gfCNCPoint1[4843] = {X 83.0240, Y 40.8731, Z -1.3333, A 0.000, B 0.000, C 0.000 }
gfCNCPoint1[4844] = {X 83.0237, Y 16.3120, Z -1.3333, A 0.000, B 0.000, C 0.000 }
gfCNCPoint1[4845] = {X 82.3786, Y 15.6228, Z -1.3333, A 0.000, B 0.000, C 0.000 }
gfCNCPoint1[4846] = {X 81.8954, Y 14.8118, Z -1.3333, A 0.000, B 0.000, C 0.000 }
gfCNCPoint1[4847] = {X 81.5963, Y 13.9165, Z -1.3333, A 0.000, B 0.000, C 0.000 }
gfCNCPoint1[4848] = {X 81.4951, Y 12.9779, Z -1.3333, A 0.000, B 0.000, C 0.000 }
gfCNCPoint1[4849] = {X 81.4951, Y 12.1868, Z -1.3333, A 0.000, B 0.000, C 0.000 }
gfCNCPoint1[4850] = {X 81.5776, Y 11.3388, Z -1.3333, A 0.000, B 0.000, C 0.000 }
gfCNCPoint1[4851] = {X 81.8219, Y 10.5227, Z -1.3333, A 0.000, B 0.000, C 0.000 }
gfCNCPoint1[4852] = {X 82.2190, Y 9.7689, Z -1.3333, A 0.000, B 0.000, C 0.000 }
gfCNCPoint1[4853] = {X 81.8180, Y 9.5051, Z -1.3333, A 0.000, B 0.000, C 0.000 }
gfCNCPoint1[4854] = {X 68.9232, Y 9.5051, Z -1.3333, A 0.000, B 0.000, C 0.000 }
gfCNCPoint1[4855] = {X 69.1905, Y 10.7210, Z -1.3333, A 0.000, B 0.000, C 0.000 }
gfCNCPoint1[4856] = {X 69.2995, Y 11.9611, Z -1.3333, A 0.000, B 0.000, C 0.000 }
gfCNCPoint1[4857] = {X 69.3015, Y 12.0739, Z -1.3333, A 0.000, B 0.000, C 0.000 }
gfCNCPoint1[4858] = {X 69.3021, Y 12.1868, Z -1.3333, A 0.000, B 0.000, C 0.000 }
gfCNCPoint1[4859] = {X 69.3017, Y 13.0686, Z -1.3333, A 0.000, B 0.000, C 0.000 }
gfCNCPoint1[4860] = {X 69.2131, Y 14.2875, Z -1.3333, A 0.000, B 0.000, C 0.000 }
gfCNCPoint1[4861] = {X 68.9717, Y 15.4855, Z -1.3333, A 0.000, B 0.000, C 0.000 }
gfCNCPoint1[4862] = {X 73.2474, Y 26.9301, Z -1.3333, A 0.000, B 0.000, C 0.000 }
gfCNCPoint1[4863] = {X 77.7438, Y 25.2502, Z -1.3333, A 0.000, B 0.000, C 0.000 }
gfCNCPoint1[4864] = {X 77.7437, Y 18.1989, Z -1.3333, A 0.000, B 0.000, C 0.000 }
gfCNCPoint1[4865] = {X 77.0787, Y 16.9748, Z -1.3333, A 0.000, B 0.000, C 0.000 }
gfCNCPoint1[4866] = {X 76.5963, Y 15.6678, Z -1.3333, A 0.000, B 0.000, C 0.000 }
gfCNCPoint1[4867] = {X 76.3065, Y 14.3051, Z -1.3333, A 0.000, B 0.000, C 0.000 }
gfCNCPoint1[4868] = {X 74.0412, Y 14.3051, Z -1.3333, A 0.000, B 0.000, C 0.000 }
gfCNCPoint1[4869] = {X 73.9997, Y 14.6975, Z -1.3333, A 0.000, B 0.000, C 0.000 }
gfCNCPoint1[4870] = {X 73.9475, Y 15.0886, Z -1.3333, A 0.000, B 0.000, C 0.000 }
gfCNCPoint1[4871] = {X 77.7438, Y 25.2502, Z -1.3333, A 0.000, B 0.000, C 0.000 }
gfCNCPoint1[4872] = {X 75.4956, Y 26.0902, Z -1.3333, A 0.000, B 0.000, C 0.000 }
gfCNCPoint1[4873] = {X 78.9539, Y 35.3470, Z -1.3333, A 0.000, B 0.000, C 0.000 }
gfCNCPoint1[4874] = {X 79.5719, Y 35.9625, Z -1.3333, A 0.000, B 0.000, C 0.000 }
gfCNCPoint1[4875] = {X 80.1440, Y 36.6209, Z -1.3333, A 0.000, B 0.000, C 0.000 }
gfCNCPoint1[4876] = {X 80.1437, Y 17.4412, Z -1.3333, A 0.000, B 0.000, C 0.000 }
gfCNCPoint1[4877] = {X 79.4950, Y 16.4475, Z -1.3333, A 0.000, B 0.000, C 0.000 }
gfCNCPoint1[4878] = {X 79.0163, Y 15.3615, Z -1.3333, A 0.000, B 0.000, C 0.000 }
gfCNCPoint1[4879] = {X 78.7204, Y 14.2122, Z -1.3333, A 0.000, B 0.000, C 0.000 }
gfCNCPoint1[4880] = {X 78.6153, Y 13.0301, Z -1.3333, A 0.000, B 0.000, C 0.000 }
gfCNCPoint1[4881] = {X 78.6151, Y 12.1868, Z -1.3333, A 0.000, B 0.000, C 0.000 }
gfCNCPoint1[4882] = {X 78.6164, Y 12.0459, Z -1.3333, A 0.000, B 0.000, C 0.000 }
gfCNCPoint1[4883] = {X 78.6205, Y 11.9051, Z -1.3333, A 0.000, B 0.000, C 0.000 }
gfCNCPoint1[4884] = {X 71.6988, Y 11.9051, Z -1.3333, A 0.000, B 0.000, C 0.000 }
gfCNCPoint1[4885] = {X 71.7013, Y 12.0460, Z -1.3333, A 0.000, B 0.000, C 0.000 }
gfCNCPoint1[4886] = {X 71.7021, Y 12.1868, Z -1.3333, A 0.000, B 0.000, C 0.000 }
gfCNCPoint1[4887] = {X 71.7016, Y 13.0911, Z -1.3333, A 0.000, B 0.000, C 0.000 }
gfCNCPoint1[4888] = {X 71.6389, Y 14.2118, Z -1.3333, A 0.000, B 0.000, C 0.000 }
gfCNCPoint1[4889] = {X 71.4726, Y 15.3218, Z -1.3333, A 0.000, B 0.000, C 0.000 }
gfCNCPoint1[4890] = {X 75.4956, Y 26.0902, Z -1.3333, A 0.000, B 0.000, C 0.000 }
gfCNCPoint1[4891] = {X 73.2474, Y 26.9301, Z -1.3333, A 0.000, B 0.000, C 0.000 }
gfCNCPoint1[4892] = {X 76.9168, Y 36.7519, Z -1.3333, A 0.000, B 0.000, C 0.000 }
gfCNCPoint1[4893] = {X 77.6311, Y 37.4061, Z -1.3333, A 0.000, B 0.000, C 0.000 }
gfCNCPoint1[4894] = {X 78.2765, Y 38.1284, Z -1.3333, A 0.000, B 0.000, C 0.000 }
gfCNCPoint1[4895] = {X 79.0237, Y 39.1932, Z -1.3333, A 0.000, B 0.000, C 0.000 }
gfCNCPoint1[4896] = {X 79.6214, Y 40.3484, Z -1.3333, A 0.000, B 0.000, C 0.000 }
gfCNCPoint1[4897] = {X 80.0588, Y 41.5734, Z -1.3333, A 0.000, B 0.000, C 0.000 }
gfCNCPoint1[4898] = {X 80.3281, Y 42.8460, Z -1.3333, A 0.000, B 0.000, C 0.000 }
gfCNCPoint1[4899] = {X 80.4242, Y 44.1432, Z -1.3333, A 0.000, B 0.000, C 0.000 }
gfCNCPoint1[4900] = {X 80.4245, Y 45.0000, Z -1.3333, A 0.000, B 0.000, C 0.000 }
gfCNCPoint1[4901] = {X 80.3511, Y 46.1898, Z -1.3333, A 0.000, B 0.000, C 0.000 }
gfCNCPoint1[4902] = {X 80.1320, Y 47.3615, Z -1.3333, A 0.000, B 0.000, C 0.000 }
gfCNCPoint1[4903] = {X 79.7706, Y 48.4974, Z -1.3333, A 0.000, B 0.000, C 0.000 }
gfCNCPoint1[4904] = {X 79.2722, Y 49.5803, Z -1.3333, A 0.000, B 0.000, C 0.000 }
gfCNCPoint1[4905] = {X 78.4688, Y 50.8341, Z -1.3333, A 0.000, B 0.000, C 0.000 }
gfCNCPoint1[4906] = {X 77.4826, Y 51.9498, Z -1.3333, A 0.000, B 0.000, C 0.000 }
gfCNCPoint1[4907] = {X 76.3369, Y 52.9011, Z -1.3333, A 0.000, B 0.000, C 0.000 }
gfCNCPoint1[4908] = {X 75.0589, Y 53.6653, Z -1.3333, A 0.000, B 0.000, C 0.000 }
gfCNCPoint1[4909] = {X 73.6787, Y 54.2246, Z -1.3333, A 0.000, B 0.000, C 0.000 }
gfCNCPoint1[4910] = {X 72.2292, Y 54.5655, Z -1.3333, A 0.000, B 0.000, C 0.000 }
gfCNCPoint1[4911] = {X 70.7445, Y 54.6800, Z -1.3333, A 0.000, B 0.000, C 0.000 }
gfCNCPoint1[4912] = {X 64.1851, Y 54.6800, Z -1.3333, A 0.000, B 0.000, C 0.000 }
gfCNCPoint1[4913] = {X 62.7229, Y 54.5689, Z -1.3333, A 0.000, B 0.000, C 0.000 }
gfCNCPoint1[4914] = {X 61.2943, Y 54.2383, Z -1.3333, A 0.000, B 0.000, C 0.000 }
gfCNCPoint1[4915] = {X 59.9320, Y 53.6956, Z -1.3333, A 0.000, B 0.000, C 0.000 }
gfCNCPoint1[4916] = {X 58.6673, Y 52.9534, Z -1.3333, A 0.000, B 0.000, C 0.000 }
gfCNCPoint1[4917] = {X 57.5293, Y 52.0286, Z -1.3333, A 0.000, B 0.000, C 0.000 }
gfCNCPoint1[4918] = {X 56.6337, Y 51.0563, Z -1.3333, A 0.000, B 0.000, C 0.000 }
gfCNCPoint1[4919] = {X 55.8790, Y 49.9710, Z -1.3333, A 0.000, B 0.000, C 0.000 }
gfCNCPoint1[4920] = {X 55.1243, Y 51.0563, Z -1.3333, A 0.000, B 0.000, C 0.000 }
gfCNCPoint1[4921] = {X 54.2288, Y 52.0286, Z -1.3333, A 0.000, B 0.000, C 0.000 }
gfCNCPoint1[4922] = {X 53.0907, Y 52.9534, Z -1.3333, A 0.000, B 0.000, C 0.000 }
gfCNCPoint1[4923] = {X 51.8261, Y 53.6956, Z -1.3333, A 0.000, B 0.000, C 0.000 }
gfCNCPoint1[4924] = {X 50.4638, Y 54.2383, Z -1.3333, A 0.000, B 0.000, C 0.000 }
gfCNCPoint1[4925] = {X 49.0351, Y 54.5689, Z -1.3333, A 0.000, B 0.000, C 0.000 }
gfCNCPoint1[4926] = {X 47.5729, Y 54.6800, Z -1.3333, A 0.000, B 0.000, C 0.000 }
gfCNCPoint1[4927] = {X 40.6393, Y 54.6800, Z -1.3333, A 0.000, B 0.000, C 0.000 }
gfCNCPoint1[4928] = {X 39.2448, Y 54.5790, Z -1.3333, A 0.000, B 0.000, C 0.000 }
gfCNCPoint1[4929] = {X 37.8793, Y 54.2782, Z -1.3333, A 0.000, B 0.000, C 0.000 }
gfCNCPoint1[4930] = {X 36.5715, Y 53.7838, Z -1.3333, A 0.000, B 0.000, C 0.000 }
gfCNCPoint1[4931] = {X 35.3485, Y 53.1062, Z -1.3333, A 0.000, B 0.000, C 0.000 }
gfCNCPoint1[4932] = {X 33.9156, Y 54.1337, Z -1.3333, A 0.000, B 0.000, C 0.000 }
gfCNCPoint1[4933] = {X 32.3650, Y 54.9732, Z -1.3333, A 0.000, B 0.000, C 0.000 }
gfCNCPoint1[4934] = {X 30.7213, Y 55.6115, Z -1.3333, A 0.000, B 0.000, C 0.000 }
gfCNCPoint1[4935] = {X 29.0105, Y 56.0384, Z -1.3333, A 0.000, B 0.000, C 0.000 }
gfCNCPoint1[4936] = {X 27.2597, Y 56.2471, Z -1.3333, A 0.000, B 0.000, C 0.000 }
gfCNCPoint1[4937] = {X 25.4108, Y 57.0591, Z -1.3333, A 0.000, B 0.000, C 0.000 }
gfCNCPoint1[4938] = {X 23.5216, Y 57.7721, Z -1.3333, A 0.000, B 0.000, C 0.000 }
gfCNCPoint1[4939] = {X 21.5973, Y 58.3841, Z -1.3333, A 0.000, B 0.000, C 0.000 }
gfCNCPoint1[4940] = {X 21.0307, Y 58.5413, Z -1.3333, A 0.000, B 0.000, C 0.000 }
gfCNCPoint1[4941] = {X 18.7673, Y 59.0805, Z -1.3333, A 0.000, B 0.000, C 0.000 }
gfCNCPoint1[4942] = {X 16.4706, Y 59.4536, Z -1.3333, A 0.000, B 0.000, C 0.000 }
gfCNCPoint1[4943] = {X 14.1529, Y 59.6585, Z -1.3333, A 0.000, B 0.000, C 0.000 }
gfCNCPoint1[4944] = {X 11.8264, Y 59.6941, Z -1.3333, A 0.000, B 0.000, C 0.000 }
gfCNCPoint1[4945] = {X 9.5035, Y 59.5603, Z -1.3333, A 0.000, B 0.000, C 0.000 }
gfCNCPoint1[4946] = {X 9.5035, Y 90.4949, Z -1.3333, A 0.000, B 0.000, C 0.000 }
gfCNCPoint1[4947] = {X 114.8635, Y 90.4949, Z -1.3333, A 0.000, B 0.000, C 0.000 }
gfCNCPoint1[4948] = {X 115.7480, Y 89.2990, Z -1.3333, A 0.000, B 0.000, C 0.000 }
gfCNCPoint1[4949] = {X 116.7726, Y 88.2208, Z -1.3333, A 0.000, B 0.000, C 0.000 }
gfCNCPoint1[4950] = {X 117.9221, Y 87.2767, Z -1.3333, A 0.000, B 0.000, C 0.000 }
gfCNCPoint1[4951] = {X 119.1788, Y 86.4811, Z -1.3333, A 0.000, B 0.000, C 0.000 }
gfCNCPoint1[4952] = {X 120.5238, Y 85.8459, Z -1.3333, A 0.000, B 0.000, C 0.000 }
gfCNCPoint1[4953] = {X 121.9366, Y 85.3808, Z -1.3333, A 0.000, B 0.000, C 0.000 }
gfCNCPoint1[4954] = {X 123.3959, Y 85.0929, Z -1.3333, A 0.000, B 0.000, C 0.000 }
gfCNCPoint1[4955] = {X 123.5628, Y 84.9132, Z -1.3333, A 0.000, B 0.000, C 0.000 }
gfCNCPoint1[4956] = {X 123.7278, Y 84.7318, Z -1.3333, A 0.000, B 0.000, C 0.000 }
gfCNCPoint1[4957] = {X 147.2181, Y 58.9362, Z -1.3333, A 0.000, B 0.000, C 0.000 }
gfCNCPoint1[4958] = {X 147.2180, Y 58.0000, Z -1.3333, A 0.000, B 0.000, C 0.000 }
gfCNCPoint1[4959] = {X 147.2987, Y 56.6058, Z -1.3333, A 0.000, B 0.000, C 0.000 }
gfCNCPoint1[4960] = {X 147.5398, Y 55.2303, Z -1.3333, A 0.000, B 0.000, C 0.000 }
gfCNCPoint1[4961] = {X 148.0022, Y 53.7185, Z -1.3333, A 0.000, B 0.000, C 0.000 }
gfCNCPoint1[4962] = {X 148.6580, Y 52.2800, Z -1.3333, A 0.000, B 0.000, C 0.000 }
gfCNCPoint1[4963] = {X 143.0396, Y 52.2800, Z -1.3333, A 0.000, B 0.000, C 0.000 }
gfCNCPoint1[4964] = {X 141.7807, Y 52.1703, Z -1.3333, A 0.000, B 0.000, C 0.000 }
gfCNCPoint1[4965] = {X 140.5597, Y 51.8446, Z -1.3333, A 0.000, B 0.000, C 0.000 }
gfCNCPoint1[4966] = {X 139.4134, Y 51.3126, Z -1.3333, A 0.000, B 0.000, C 0.000 }
gfCNCPoint1[4967] = {X 138.3764, Y 50.5904, Z -1.3333, A 0.000, B 0.000, C 0.000 }
gfCNCPoint1[4968] = {X 137.4799, Y 49.6998, Z -1.3333, A 0.000, B 0.000, C 0.000 }
gfCNCPoint1[4969] = {X 136.7509, Y 48.6675, Z -1.3333, A 0.000, B 0.000, C 0.000 }
gfCNCPoint1[4970] = {X 136.2114, Y 47.5248, Z -1.3333, A 0.000, B 0.000, C 0.000 }
gfCNCPoint1[4971] = {X 135.8777, Y 46.3059, Z -1.3333, A 0.000, B 0.000, C 0.000 }
gfCNCPoint1[4972] = {X 135.7598, Y 45.0477, Z -1.3333, A 0.000, B 0.000, C 0.000 }
gfCNCPoint1[4973] = {X 135.7601, Y 44.1247, Z -1.3333, A 0.000, B 0.000, C 0.000 }
gfCNCPoint1[4974] = {X 135.8408, Y 43.1249, Z -1.3333, A 0.000, B 0.000, C 0.000 }
gfCNCPoint1[4975] = {X 136.0581, Y 42.1457, Z -1.3333, A 0.000, B 0.000, C 0.000 }
gfCNCPoint1[4976] = {X 138.3597, Y 42.8258, Z -1.3333, A 0.000, B 0.000, C 0.000 }
gfCNCPoint1[4977] = {X 138.6721, Y 42.0319, Z -1.3333, A 0.000, B 0.000, C 0.000 }
gfCNCPoint1[4978] = {X 139.1179, Y 41.3046, Z -1.3333, A 0.000, B 0.000, C 0.000 }
gfCNCPoint1[4979] = {X 139.6836, Y 40.6660, Z -1.3333, A 0.000, B 0.000, C 0.000 }
gfCNCPoint1[4980] = {X 139.6836, Y 20.4363, Z -1.3333, A 0.000, B 0.000, C 0.000 }
gfCNCPoint1[4981] = {X 137.7113, Y 20.4357, Z -1.3333, A 0.000, B 0.000, C 0.000 }
gfCNCPoint1[4982] = {X 137.0006, Y 21.1817, Z -1.3333, A 0.000, B 0.000, C 0.000 }
gfCNCPoint1[4983] = {X 136.1491, Y 21.7619, Z -1.3333, A 0.000, B 0.000, C 0.000 }
gfCNCPoint1[4984] = {X 135.4282, Y 22.0767, Z -1.3333, A 0.000, B 0.000, C 0.000 }
gfCNCPoint1[4985] = {X 134.6660, Y 22.2715, Z -1.3333, A 0.000, B 0.000, C 0.000 }
gfCNCPoint1[4986] = {X 133.8824, Y 22.3414, Z -1.3333, A 0.000, B 0.000, C 0.000 }
gfCNCPoint1[4987] = {X 133.2006, Y 22.3415, Z -1.3333, A 0.000, B 0.000, C 0.000 }
gfCNCPoint1[4988] = {X 132.2486, Y 22.2478, Z -1.3333, A 0.000, B 0.000, C 0.000 }
gfCNCPoint1[4989] = {X 131.3331, Y 21.9701, Z -1.3333, A 0.000, B 0.000, C 0.000 }
gfCNCPoint1[4990] = {X 130.4895, Y 21.5191, Z -1.3333, A 0.000, B 0.000, C 0.000 }
gfCNCPoint1[4991] = {X 129.7500, Y 20.9122, Z -1.3333, A 0.000, B 0.000, C 0.000 }
gfCNCPoint1[4992] = {X 129.1431, Y 20.1727, Z -1.3333, A 0.000, B 0.000, C 0.000 }
gfCNCPoint1[4993] = {X 128.6921, Y 19.3290, Z -1.3333, A 0.000, B 0.000, C 0.000 }
gfCNCPoint1[4994] = {X 128.4144, Y 18.4136, Z -1.3333, A 0.000, B 0.000, C 0.000 }
gfCNCPoint1[4995] = {X 128.3206, Y 17.4615, Z -1.3333, A 0.000, B 0.000, C 0.000 }
gfCNCPoint1[4996] = {X 128.3206, Y 10.4835, Z -1.3333, A 0.000, B 0.000, C 0.000 }
gfCNCPoint1[4997] = {X 128.3317, Y 10.1548, Z -1.3333, A 0.000, B 0.000, C 0.000 }
gfCNCPoint1[4998] = {X 128.3649, Y 9.8277, Z -1.3333, A 0.000, B 0.000, C 0.000 }
gfCNCPoint1[4999] = {X 128.6078, Y 8.8342, Z -1.3333, A 0.000, B 0.000, C 0.000 }
gfCNCPoint1[5000] = {X 129.0524, Y 7.9132, Z -1.3333, A 0.000, B 0.000, C 0.000 }
gfCNCPoint1[5001] = {X 129.6792, Y 7.1051, Z -1.3333, A 0.000, B 0.000, C 0.000 }
gfCNCPoint1[5002] = {X 130.0255, Y 7.4374, Z -1.3333, A 0.000, B 0.000, C 0.000 }
gfCNCPoint1[5003] = {X 130.6996, Y 6.8635, Z -1.3333, A 0.000, B 0.000, C 0.000 }
gfCNCPoint1[5004] = {X 131.4748, Y 6.4361, Z -1.3333, A 0.000, B 0.000, C 0.000 }
gfCNCPoint1[5005] = {X 132.3199, Y 6.1726, Z -1.3333, A 0.000, B 0.000, C 0.000 }
gfCNCPoint1[5006] = {X 133.2007, Y 6.0835, Z -1.3333, A 0.000, B 0.000, C 0.000 }
gfCNCPoint1[5007] = {X 133.8874, Y 6.0837, Z -1.3333, A 0.000, B 0.000, C 0.000 }
gfCNCPoint1[5008] = {X 134.7192, Y 6.1718, Z -1.3333, A 0.000, B 0.000, C 0.000 }
gfCNCPoint1[5009] = {X 135.5192, Y 6.4156, Z -1.3333, A 0.000, B 0.000, C 0.000 }
gfCNCPoint1[5010] = {X 136.2587, Y 6.8064, Z -1.3333, A 0.000, B 0.000, C 0.000 }
gfCNCPoint1[5011] = {X 136.9108, Y 7.3301, Z -1.3333, A 0.000, B 0.000, C 0.000 }
gfCNCPoint1[5012] = {X 137.4521, Y 7.9677, Z -1.3333, A 0.000, B 0.000, C 0.000 }
gfCNCPoint1[5013] = {X 155.0706, Y 7.9677, Z -1.3333, A 0.000, B 0.000, C 0.000 }
gfCNCPoint1[5014] = {X 155.6184, Y 7.3238, Z -1.3333, A 0.000, B 0.000, C 0.000 }
gfCNCPoint1[5015] = {X 156.2792, Y 6.7965, Z -1.3333, A 0.000, B 0.000, C 0.000 }
gfCNCPoint1[5016] = {X 157.0287, Y 6.4053, Z -1.3333, A 0.000, B 0.000, C 0.000 }
gfCNCPoint1[5017] = {X 157.8391, Y 6.1647, Z -1.3333, A 0.000, B 0.000, C 0.000 }
gfCNCPoint1[5018] = {X 158.6806, Y 6.0835, Z -1.3333, A 0.000, B 0.000, C 0.000 }
gfCNCPoint1[5019] = {X 159.3791, Y 6.0839, Z -1.3333, A 0.000, B 0.000, C 0.000 }
gfCNCPoint1[5020] = {X 160.3488, Y 6.2050, Z -1.3333, A 0.000, B 0.000, C 0.000 }
gfCNCPoint1[5021] = {X 161.2678, Y 6.5371, Z -1.3333, A 0.000, B 0.000, C 0.000 }
gfCNCPoint1[5022] = {X 162.0908, Y 7.0639, Z -1.3333, A 0.000, B 0.000, C 0.000 }
gfCNCPoint1[5023] = {X 162.7773, Y 7.7593, Z -1.3333, A 0.000, B 0.000, C 0.000 }
gfCNCPoint1[5024] = {X 163.2934, Y 8.5891, Z -1.3333, A 0.000, B 0.000, C 0.000 }
gfCNCPoint1[5025] = {X 163.6136, Y 9.5124, Z -1.3333, A 0.000, B 0.000, C 0.000 }
gfCNCPoint1[5026] = {X 163.7221, Y 10.4835, Z -1.3333, A 0.000, B 0.000, C 0.000 }
gfCNCPoint1[5027] = {X 163.7221, Y 17.4615, Z -1.3333, A 0.000, B 0.000, C 0.000 }
gfCNCPoint1[5028] = {X 163.6118, Y 18.4406, Z -1.3333, A 0.000, B 0.000, C 0.000 }
gfCNCPoint1[5029] = {X 163.2863, Y 19.3706, Z -1.3333, A 0.000, B 0.000, C 0.000 }
gfCNCPoint1[5030] = {X 162.7621, Y 20.2049, Z -1.3333, A 0.000, B 0.000, C 0.000 }
gfCNCPoint1[5031] = {X 162.0654, Y 20.9016, Z -1.3333, A 0.000, B 0.000, C 0.000 }
gfCNCPoint1[5032] = {X 161.2312, Y 21.4258, Z -1.3333, A 0.000, B 0.000, C 0.000 }
gfCNCPoint1[5033] = {X 160.3011, Y 21.7512, Z -1.3333, A 0.000, B 0.000, C 0.000 }
gfCNCPoint1[5034] = {X 159.3221, Y 21.8615, Z -1.3333, A 0.000, B 0.000, C 0.000 }
gfCNCPoint1[5035] = {X 158.6785, Y 21.8615, Z -1.3333, A 0.000, B 0.000, C 0.000 }
gfCNCPoint1[5036] = {X 157.8332, Y 21.7759, Z -1.3333, A 0.000, B 0.000, C 0.000 }
gfCNCPoint1[5037] = {X 157.0197, Y 21.5308, Z -1.3333, A 0.000, B 0.000, C 0.000 }
gfCNCPoint1[5038] = {X 156.2678, Y 21.1352, Z -1.3333, A 0.000, B 0.000, C 0.000 }
gfCNCPoint1[5039] = {X 155.6049, Y 20.6037, Z -1.3333, A 0.000, B 0.000, C 0.000 }
gfCNCPoint1[5040] = {X 155.0555, Y 19.9556, Z -1.3333, A 0.000, B 0.000, C 0.000 }
gfCNCPoint1[5041] = {X 152.3555, Y 19.9571, Z -1.3333, A 0.000, B 0.000, C 0.000 }
gfCNCPoint1[5042] = {X 152.3538, Y 40.8427, Z -1.3333, A 0.000, B 0.000, C 0.000 }
gfCNCPoint1[5043] = {X 152.8077, Y 41.3321, Z -1.3333, A 0.000, B 0.000, C 0.000 }
gfCNCPoint1[5044] = {X 152.8988, Y 41.4411, Z -1.3333, A 0.000, B 0.000, C 0.000 }
gfCNCPoint1[5045] = {X 153.4331, Y 42.2816, Z -1.3333, A 0.000, B 0.000, C 0.000 }
gfCNCPoint1[5046] = {X 153.7667, Y 43.2199, Z -1.3333, A 0.000, B 0.000, C 0.000 }
gfCNCPoint1[5047] = {X 153.8831, Y 44.2089, Z -1.3333, A 0.000, B 0.000, C 0.000 }
gfCNCPoint1[5048] = {X 153.8829, Y 45.0423, Z -1.3333, A 0.000, B 0.000, C 0.000 }
gfCNCPoint1[5049] = {X 153.7646, Y 46.0144, Z -1.3333, A 0.000, B 0.000, C 0.000 }
gfCNCPoint1[5050] = {X 153.4342, Y 46.9363, Z -1.3333, A 0.000, B 0.000, C 0.000 }
gfCNCPoint1[5051] = {X 152.9080, Y 47.7622, Z -1.3333, A 0.000, B 0.000, C 0.000 }
gfCNCPoint1[5052] = {X 152.2123, Y 48.4513, Z -1.3333, A 0.000, B 0.000, C 0.000 }
gfCNCPoint1[5053] = {X 151.3813, Y 48.9695, Z -1.3333, A 0.000, B 0.000, C 0.000 }
gfCNCPoint1[5054] = {X 150.4563, Y 49.2910, Z -1.3333, A 0.000, B 0.000, C 0.000 }
gfCNCPoint1[5055] = {X 149.4831, Y 49.4000, Z -1.3333, A 0.000, B 0.000, C 0.000 }
gfCNCPoint1[5056] = {X 143.0396, Y 49.4000, Z -1.3333, A 0.000, B 0.000, C 0.000 }
gfCNCPoint1[5057] = {X 142.0605, Y 49.2897, Z -1.3333, A 0.000, B 0.000, C 0.000 }
gfCNCPoint1[5058] = {X 141.1305, Y 48.9643, Z -1.3333, A 0.000, B 0.000, C 0.000 }
gfCNCPoint1[5059] = {X 140.2963, Y 48.4400, Z -1.3333, A 0.000, B 0.000, C 0.000 }
gfCNCPoint1[5060] = {X 139.5996, Y 47.7433, Z -1.3333, A 0.000, B 0.000, C 0.000 }
gfCNCPoint1[5061] = {X 139.0754, Y 46.9091, Z -1.3333, A 0.000, B 0.000, C 0.000 }
gfCNCPoint1[5062] = {X 138.7499, Y 45.9790, Z -1.3333, A 0.000, B 0.000, C 0.000 }
gfCNCPoint1[5063] = {X 138.6396, Y 44.9999, Z -1.3333, A 0.000, B 0.000, C 0.000 }
gfCNCPoint1[5064] = {X 138.6400, Y 44.1483, Z -1.3333, A 0.000, B 0.000, C 0.000 }
gfCNCPoint1[5065] = {X 138.7505, Y 43.2275, Z -1.3333, A 0.000, B 0.000, C 0.000 }
gfCNCPoint1[5066] = {X 139.0514, Y 42.3503, Z -1.3333, A 0.000, B 0.000, C 0.000 }
gfCNCPoint1[5067] = {X 139.5295, Y 41.5556, Z -1.3333, A 0.000, B 0.000, C 0.000 }
gfCNCPoint1[5068] = {X 140.1636, Y 40.8789, Z -1.3333, A 0.000, B 0.000, C 0.000 }
gfCNCPoint1[5069] = {X 140.1636, Y 19.9565, Z -1.3333, A 0.000, B 0.000, C 0.000 }
gfCNCPoint1[5070] = {X 137.4672, Y 19.9556, Z -1.3333, A 0.000, B 0.000, C 0.000 }
gfCNCPoint1[5071] = {X 136.9195, Y 20.6065, Z -1.3333, A 0.000, B 0.000, C 0.000 }
gfCNCPoint1[5072] = {X 136.2568, Y 21.1399, Z -1.3333, A 0.000, B 0.000, C 0.000 }
gfCNCPoint1[5073] = {X 135.5039, Y 21.5358, Z -1.3333, A 0.000, B 0.000, C 0.000 }
gfCNCPoint1[5074] = {X 134.6888, Y 21.7793, Z -1.3333, A 0.000, B 0.000, C 0.000 }
gfCNCPoint1[5075] = {X 133.8421, Y 21.8615, Z -1.3333, A 0.000, B 0.000, C 0.000 }
gfCNCPoint1[5076] = {X 133.2006, Y 21.8615, Z -1.3333, A 0.000, B 0.000, C 0.000 }
gfCNCPoint1[5077] = {X 132.2215, Y 21.7512, Z -1.3333, A 0.000, B 0.000, C 0.000 }
gfCNCPoint1[5078] = {X 131.2916, Y 21.4258, Z -1.3333, A 0.000, B 0.000, C 0.000 }
gfCNCPoint1[5079] = {X 130.4573, Y 20.9016, Z -1.3333, A 0.000, B 0.000, C 0.000 }
gfCNCPoint1[5080] = {X 129.7606, Y 20.2049, Z -1.3333, A 0.000, B 0.000, C 0.000 }
gfCNCPoint1[5081] = {X 129.2364, Y 19.3706, Z -1.3333, A 0.000, B 0.000, C 0.000 }
gfCNCPoint1[5082] = {X 128.9110, Y 18.4406, Z -1.3333, A 0.000, B 0.000, C 0.000 }
gfCNCPoint1[5083] = {X 128.8006, Y 17.4615, Z -1.3333, A 0.000, B 0.000, C 0.000 }
gfCNCPoint1[5084] = {X 128.8006, Y 10.4835, Z -1.3333, A 0.000, B 0.000, C 0.000 }
gfCNCPoint1[5085] = {X 128.8808, Y 9.6475, Z -1.3333, A 0.000, B 0.000, C 0.000 }
gfCNCPoint1[5086] = {X 129.1183, Y 8.8419, Z -1.3333, A 0.000, B 0.000, C 0.000 }
gfCNCPoint1[5087] = {X 129.5046, Y 8.0962, Z -1.3333, A 0.000, B 0.000, C 0.000 }
gfCNCPoint1[5088] = {X 130.0255, Y 7.4374, Z -1.3333, A 0.000, B 0.000, C 0.000 }
gfCNCPoint1[5089] = {X 129.6792, Y 7.1051, Z -1.3333, A 0.000, B 0.000, C 0.000 }
gfCNCPoint1[5090] = {X 102.4337, Y 7.1051, Z -1.3333, A 0.000, B 0.000, C 0.000 }
gfCNCPoint1[5091] = {X 102.4337, Y 11.9051, Z -1.3333, A 0.000, B 0.000, C 0.000 }
gfCNCPoint1[5092] = {X 101.3242, Y 11.9051, Z -1.3333, A 0.000, B 0.000, C 0.000 }
gfCNCPoint1[5093] = {X 101.3283, Y 12.0459, Z -1.3333, A 0.000, B 0.000, C 0.000 }
gfCNCPoint1[5094] = {X 101.3297, Y 12.1868, Z -1.3333, A 0.000, B 0.000, C 0.000 }
gfCNCPoint1[5095] = {X 101.3293, Y 13.0462, Z -1.3333, A 0.000, B 0.000, C 0.000 }
gfCNCPoint1[5096] = {X 101.2273, Y 14.1946, Z -1.3333, A 0.000, B 0.000, C 0.000 }
gfCNCPoint1[5097] = {X 100.9452, Y 15.3125, Z -1.3333, A 0.000, B 0.000, C 0.000 }
gfCNCPoint1[5098] = {X 101.0384, Y 15.5444, Z -1.3333, A 0.000, B 0.000, C 0.000 }
gfCNCPoint1[5099] = {X 101.8683, Y 17.6021, Z -1.3333, A 0.000, B 0.000, C 0.000 }
gfCNCPoint1[5100] = {X 102.8007, Y 15.2768, Z -1.3333, A 0.000, B 0.000, C 0.000 }
gfCNCPoint1[5101] = {X 102.5275, Y 14.1756, Z -1.3333, A 0.000, B 0.000, C 0.000 }
gfCNCPoint1[5102] = {X 102.4286, Y 13.0453, Z -1.3333, A 0.000, B 0.000, C 0.000 }
gfCNCPoint1[5103] = {X 102.4283, Y 12.1868, Z -1.3333, A 0.000, B 0.000, C 0.000 }
gfCNCPoint1[5104] = {X 102.4296, Y 12.0459, Z -1.3333, A 0.000, B 0.000, C 0.000 }
gfCNCPoint1[5105] = {X 102.4337, Y 11.9051, Z -1.3333, A 0.000, B 0.000, C 0.000 }
gfCNCPoint1[5106] = {X 102.4337, Y 9.5051, Z -1.3333, A 0.000, B 0.000, C 0.000 }
gfCNCPoint1[5107] = {X 98.1268, Y 9.5051, Z -1.3333, A 0.000, B 0.000, C 0.000 }
gfCNCPoint1[5108] = {X 98.5430, Y 10.2830, Z -1.3333, A 0.000, B 0.000, C 0.000 }
gfCNCPoint1[5109] = {X 98.8123, Y 11.1231, Z -1.3333, A 0.000, B 0.000, C 0.000 }
gfCNCPoint1[5110] = {X 98.9260, Y 11.9980, Z -1.3333, A 0.000, B 0.000, C 0.000 }
gfCNCPoint1[5111] = {X 98.9288, Y 12.0924, Z -1.3333, A 0.000, B 0.000, C 0.000 }
gfCNCPoint1[5112] = {X 98.9297, Y 12.1868, Z -1.3333, A 0.000, B 0.000, C 0.000 }
gfCNCPoint1[5113] = {X 98.9294, Y 13.0237, Z -1.3333, A 0.000, B 0.000, C 0.000 }
gfCNCPoint1[5114] = {X 98.8589, Y 13.8063, Z -1.3333, A 0.000, B 0.000, C 0.000 }
gfCNCPoint1[5115] = {X 98.6636, Y 14.5673, Z -1.3333, A 0.000, B 0.000, C 0.000 }
gfCNCPoint1[5116] = {X 98.3487, Y 15.2872, Z -1.3333, A 0.000, B 0.000, C 0.000 }
gfCNCPoint1[5117] = {X 98.8120, Y 16.4405, Z -1.3333, A 0.000, B 0.000, C 0.000 }
gfCNCPoint1[5118] = {X 101.8749, Y 24.0344, Z -1.3333, A 0.000, B 0.000, C 0.000 }
gfCNCPoint1[5119] = {X 105.3939, Y 15.2584, Z -1.3333, A 0.000, B 0.000, C 0.000 }
gfCNCPoint1[5120] = {X 105.0872, Y 14.5466, Z -1.3333, A 0.000, B 0.000, C 0.000 }
gfCNCPoint1[5121] = {X 104.8972, Y 13.7951, Z -1.3333, A 0.000, B 0.000, C 0.000 }
gfCNCPoint1[5122] = {X 104.8285, Y 13.0231, Z -1.3333, A 0.000, B 0.000, C 0.000 }
gfCNCPoint1[5123] = {X 104.8283, Y 12.1868, Z -1.3333, A 0.000, B 0.000, C 0.000 }
gfCNCPoint1[5124] = {X 104.8292, Y 12.0924, Z -1.3333, A 0.000, B 0.000, C 0.000 }
gfCNCPoint1[5125] = {X 104.8319, Y 11.9980, Z -1.3333, A 0.000, B 0.000, C 0.000 }
gfCNCPoint1[5126] = {X 104.9456, Y 11.1231, Z -1.3333, A 0.000, B 0.000, C 0.000 }
gfCNCPoint1[5127] = {X 105.2150, Y 10.2830, Z -1.3333, A 0.000, B 0.000, C 0.000 }
gfCNCPoint1[5128] = {X 105.6312, Y 9.5051, Z -1.3333, A 0.000, B 0.000, C 0.000 }
gfCNCPoint1[5129] = {X 102.4337, Y 9.5051, Z -1.3333, A 0.000, B 0.000, C 0.000 }
gfCNCPoint1[5130] = {X 102.4337, Y 7.1051, Z -1.3333, A 0.000, B 0.000, C 0.000 }
gfCNCPoint1[5131] = {X 64.8351, Y 7.1051, Z -1.3333, A 0.000, B 0.000, C 0.000 }
gfCNCPoint1[5132] = {X 65.5947, Y 8.0243, Z -1.3333, A 0.000, B 0.000, C 0.000 }
gfCNCPoint1[5133] = {X 66.1941, Y 9.0551, Z -1.3333, A 0.000, B 0.000, C 0.000 }
gfCNCPoint1[5134] = {X 66.6172, Y 10.1700, Z -1.3333, A 0.000, B 0.000, C 0.000 }
gfCNCPoint1[5135] = {X 66.8305, Y 11.1684, Z -1.3333, A 0.000, B 0.000, C 0.000 }
gfCNCPoint1[5136] = {X 66.9021, Y 12.1868, Z -1.3333, A 0.000, B 0.000, C 0.000 }
gfCNCPoint1[5137] = {X 66.9018, Y 13.0462, Z -1.3333, A 0.000, B 0.000, C 0.000 }
gfCNCPoint1[5138] = {X 66.7777, Y 14.3180, Z -1.3333, A 0.000, B 0.000, C 0.000 }
gfCNCPoint1[5139] = {X 66.4332, Y 15.5485, Z -1.3333, A 0.000, B 0.000, C 0.000 }
gfCNCPoint1[5140] = {X 74.9101, Y 38.2384, Z -1.3333, A 0.000, B 0.000, C 0.000 }
gfCNCPoint1[5141] = {X 75.8027, Y 38.9731, Z -1.3333, A 0.000, B 0.000, C 0.000 }
gfCNCPoint1[5142] = {X 76.5678, Y 39.8400, Z -1.3333, A 0.000, B 0.000, C 0.000 }
gfCNCPoint1[5143] = {X 77.1861, Y 40.8170, Z -1.3333, A 0.000, B 0.000, C 0.000 }
gfCNCPoint1[5144] = {X 77.6418, Y 41.8796, Z -1.3333, A 0.000, B 0.000, C 0.000 }
gfCNCPoint1[5145] = {X 77.9236, Y 43.0009, Z -1.3333, A 0.000, B 0.000, C 0.000 }
gfCNCPoint1[5146] = {X 78.0243, Y 44.1527, Z -1.3333, A 0.000, B 0.000, C 0.000 }
gfCNCPoint1[5147] = {X 78.0245, Y 45.0000, Z -1.3333, A 0.000, B 0.000, C 0.000 }
gfCNCPoint1[5148] = {X 77.9139, Y 46.2642, Z -1.3333, A 0.000, B 0.000, C 0.000 }
gfCNCPoint1[5149] = {X 77.5854, Y 47.4899, Z -1.3333, A 0.000, B 0.000, C 0.000 }
gfCNCPoint1[5150] = {X 77.0491, Y 48.6400, Z -1.3333, A 0.000, B 0.000, C 0.000 }
gfCNCPoint1[5151] = {X 76.3213, Y 49.6795, Z -1.3333, A 0.000, B 0.000, C 0.000 }
gfCNCPoint1[5152] = {X 75.4240, Y 50.5768, Z -1.3333, A 0.000, B 0.000, C 0.000 }
gfCNCPoint1[5153] = {X 74.3845, Y 51.3047, Z -1.3333, A 0.000, B 0.000, C 0.000 }
gfCNCPoint1[5154] = {X 73.2344, Y 51.8410, Z -1.3333, A 0.000, B 0.000, C 0.000 }
gfCNCPoint1[5155] = {X 72.0086, Y 52.1694, Z -1.3333, A 0.000, B 0.000, C 0.000 }
gfCNCPoint1[5156] = {X 70.7445, Y 52.2800, Z -1.3333, A 0.000, B 0.000, C 0.000 }
gfCNCPoint1[5157] = {X 64.1851, Y 52.2800, Z -1.3333, A 0.000, B 0.000, C 0.000 }
gfCNCPoint1[5158] = {X 62.9397, Y 52.1727, Z -1.3333, A 0.000, B 0.000, C 0.000 }
gfCNCPoint1[5159] = {X 61.7311, Y 51.8539, Z -1.3333, A 0.000, B 0.000, C 0.000 }
gfCNCPoint1[5160] = {X 60.5947, Y 51.3330, Z -1.3333, A 0.000, B 0.000, C 0.000 }
gfCNCPoint1[5161] = {X 59.5643, Y 50.6255, Z -1.3333, A 0.000, B 0.000, C 0.000 }
gfCNCPoint1[5162] = {X 58.6700, Y 49.7521, Z -1.3333, A 0.000, B 0.000, C 0.000 }
gfCNCPoint1[5163] = {X 57.9384, Y 48.7385, Z -1.3333, A 0.000, B 0.000, C 0.000 }
gfCNCPoint1[5164] = {X 57.3706, Y 47.5614, Z -1.3333, A 0.000, B 0.000, C 0.000 }
gfCNCPoint1[5165] = {X 57.0224, Y 46.3017, Z -1.3333, A 0.000, B 0.000, C 0.000 }
gfCNCPoint1[5166] = {X 56.9051, Y 45.0000, Z -1.3333, A 0.000, B 0.000, C 0.000 }
gfCNCPoint1[5167] = {X 56.9052, Y 44.1969, Z -1.3333, A 0.000, B 0.000, C 0.000 }
gfCNCPoint1[5168] = {X 56.9289, Y 43.6212, Z -1.3333, A 0.000, B 0.000, C 0.000 }
gfCNCPoint1[5169] = {X 56.9981, Y 43.0492, Z -1.3333, A 0.000, B 0.000, C 0.000 }
gfCNCPoint1[5170] = {X 54.7600, Y 43.0492, Z -1.3333, A 0.000, B 0.000, C 0.000 }
gfCNCPoint1[5171] = {X 54.8275, Y 43.6012, Z -1.3333, A 0.000, B 0.000, C 0.000 }
gfCNCPoint1[5172] = {X 54.8528, Y 44.1567, Z -1.3333, A 0.000, B 0.000, C 0.000 }
gfCNCPoint1[5173] = {X 54.8529, Y 45.0000, Z -1.3333, A 0.000, B 0.000, C 0.000 }
gfCNCPoint1[5174] = {X 54.7356, Y 46.3017, Z -1.3333, A 0.000, B 0.000, C 0.000 }
gfCNCPoint1[5175] = {X 54.3875, Y 47.5614, Z -1.3333, A 0.000, B 0.000, C 0.000 }
gfCNCPoint1[5176] = {X 53.8197, Y 48.7385, Z -1.3333, A 0.000, B 0.000, C 0.000 }
gfCNCPoint1[5177] = {X 53.0880, Y 49.7521, Z -1.3333, A 0.000, B 0.000, C 0.000 }
gfCNCPoint1[5178] = {X 52.1938, Y 50.6255, Z -1.3333, A 0.000, B 0.000, C 0.000 }
gfCNCPoint1[5179] = {X 51.1633, Y 51.3330, Z -1.3333, A 0.000, B 0.000, C 0.000 }
gfCNCPoint1[5180] = {X 50.0270, Y 51.8539, Z -1.3333, A 0.000, B 0.000, C 0.000 }
gfCNCPoint1[5181] = {X 48.8183, Y 52.1727, Z -1.3333, A 0.000, B 0.000, C 0.000 }
gfCNCPoint1[5182] = {X 47.5729, Y 52.2800, Z -1.3333, A 0.000, B 0.000, C 0.000 }
gfCNCPoint1[5183] = {X 40.6393, Y 52.2800, Z -1.3333, A 0.000, B 0.000, C 0.000 }
gfCNCPoint1[5184] = {X 39.4476, Y 52.1818, Z -1.3333, A 0.000, B 0.000, C 0.000 }
gfCNCPoint1[5185] = {X 38.2881, Y 51.8899, Z -1.3333, A 0.000, B 0.000, C 0.000 }
gfCNCPoint1[5186] = {X 37.1919, Y 51.4120, Z -1.3333, A 0.000, B 0.000, C 0.000 }
gfCNCPoint1[5187] = {X 36.1888, Y 50.7612, Z -1.3333, A 0.000, B 0.000, C 0.000 }
gfCNCPoint1[5188] = {X 35.3058, Y 49.9550, Z -1.3333, A 0.000, B 0.000, C 0.000 }
gfCNCPoint1[5189] = {X 34.8234, Y 50.4196, Z -1.3333, A 0.000, B 0.000, C 0.000 }
gfCNCPoint1[5190] = {X 34.3150, Y 50.8555, Z -1.3333, A 0.000, B 0.000, C 0.000 }
gfCNCPoint1[5191] = {X 33.7697, Y 51.2964, Z -1.3333, A 0.000, B 0.000, C 0.000 }
gfCNCPoint1[5192] = {X 32.5122, Y 52.1794, Z -1.3333, A 0.000, B 0.000, C 0.000 }
gfCNCPoint1[5193] = {X 31.1492, Y 52.8887, Z -1.3333, A 0.000, B 0.000, C 0.000 }
gfCNCPoint1[5194] = {X 29.7045, Y 53.4120, Z -1.3333, A 0.000, B 0.000, C 0.000 }
gfCNCPoint1[5195] = {X 28.2034, Y 53.7401, Z -1.3333, A 0.000, B 0.000, C 0.000 }
gfCNCPoint1[5196] = {X 26.6721, Y 53.8673, Z -1.3333, A 0.000, B 0.000, C 0.000 }
gfCNCPoint1[5197] = {X 24.8056, Y 54.7124, Z -1.3333, A 0.000, B 0.000, C 0.000 }
gfCNCPoint1[5198] = {X 22.8937, Y 55.4491, Z -1.3333, A 0.000, B 0.000, C 0.000 }
gfCNCPoint1[5199] = {X 20.9428, Y 56.0750, Z -1.3333, A 0.000, B 0.000, C 0.000 }
gfCNCPoint1[5200] = {X 20.3898, Y 56.2285, Z -1.3333, A 0.000, B 0.000, C 0.000 }
gfCNCPoint1[5201] = {X 18.2965, Y 56.7272, Z -1.3333, A 0.000, B 0.000, C 0.000 }
gfCNCPoint1[5202] = {X 16.1724, Y 57.0722, Z -1.3333, A 0.000, B 0.000, C 0.000 }
gfCNCPoint1[5203] = {X 14.0288, Y 57.2617, Z -1.3333, A 0.000, B 0.000, C 0.000 }
gfCNCPoint1[5204] = {X 11.8771, Y 57.2946, Z -1.3333, A 0.000, B 0.000, C 0.000 }
gfCNCPoint1[5205] = {X 9.7287, Y 57.1709, Z -1.3333, A 0.000, B 0.000, C 0.000 }
gfCNCPoint1[5206] = {X 8.7885, Y 57.0670, Z -1.3333, A 0.000, B 0.000, C 0.000 }
gfCNCPoint1[5207] = {X 7.8521, Y 56.9332, Z -1.3333, A 0.000, B 0.000, C 0.000 }
gfCNCPoint1[5208] = {X 7.4773, Y 56.8761, Z -1.3333, A 0.000, B 0.000, C 0.000 }
gfCNCPoint1[5209] = {X 7.1035, Y 56.8133, Z -1.3333, A 0.000, B 0.000, C 0.000 }
gfCNCPoint1[5210] = {X 7.1035, Y 92.8949, Z -1.3333, A 0.000, B 0.000, C 0.000 }
gfCNCPoint1[5211] = {X 116.2647, Y 92.8949, Z -1.3333, A 0.000, B 0.000, C 0.000 }
gfCNCPoint1[5212] = {X 116.9731, Y 91.6556, Z -1.3333, A 0.000, B 0.000, C 0.000 }
gfCNCPoint1[5213] = {X 117.8561, Y 90.5340, Z -1.3333, A 0.000, B 0.000, C 0.000 }
gfCNCPoint1[5214] = {X 118.8944, Y 89.5544, Z -1.3333, A 0.000, B 0.000, C 0.000 }
gfCNCPoint1[5215] = {X 120.0654, Y 88.7381, Z -1.3333, A 0.000, B 0.000, C 0.000 }
gfCNCPoint1[5216] = {X 121.3438, Y 88.1030, Z -1.3333, A 0.000, B 0.000, C 0.000 }
gfCNCPoint1[5217] = {X 122.7017, Y 87.6627, Z -1.3333, A 0.000, B 0.000, C 0.000 }
gfCNCPoint1[5218] = {X 124.1096, Y 87.4270, Z -1.3333, A 0.000, B 0.000, C 0.000 }
gfCNCPoint1[5219] = {X 124.5364, Y 87.3628, Z -1.3333, A 0.000, B 0.000, C 0.000 }
gfCNCPoint1[5220] = {X 125.0286, Y 86.8594, Z -1.3333, A 0.000, B 0.000, C 0.000 }
gfCNCPoint1[5221] = {X 125.5069, Y 86.3427, Z -1.3333, A 0.000, B 0.000, C 0.000 }
gfCNCPoint1[5222] = {X 149.6586, Y 59.8207, Z -1.3333, A 0.000, B 0.000, C 0.000 }
gfCNCPoint1[5223] = {X 149.6295, Y 59.4073, Z -1.3333, A 0.000, B 0.000, C 0.000 }
gfCNCPoint1[5224] = {X 149.6181, Y 58.9930, Z -1.3333, A 0.000, B 0.000, C 0.000 }
gfCNCPoint1[5225] = {X 149.6180, Y 58.0000, Z -1.3333, A 0.000, B 0.000, C 0.000 }
gfCNCPoint1[5226] = {X 149.6915, Y 56.8093, Z -1.3333, A 0.000, B 0.000, C 0.000 }
gfCNCPoint1[5227] = {X 149.9109, Y 55.6367, Z -1.3333, A 0.000, B 0.000, C 0.000 }
gfCNCPoint1[5228] = {X 150.2729, Y 54.5000, Z -1.3333, A 0.000, B 0.000, C 0.000 }
gfCNCPoint1[5229] = {X 150.7719, Y 53.4164, Z -1.3333, A 0.000, B 0.000, C 0.000 }
gfCNCPoint1[5230] = {X 151.5117, Y 52.2488, Z -1.3333, A 0.000, B 0.000, C 0.000 }
gfCNCPoint1[5231] = {X 152.4103, Y 51.1984, Z -1.3333, A 0.000, B 0.000, C 0.000 }
gfCNCPoint1[5232] = {X 153.4493, Y 50.2867, Z -1.3333, A 0.000, B 0.000, C 0.000 }
gfCNCPoint1[5233] = {X 154.6075, Y 49.5323, Z -1.3333, A 0.000, B 0.000, C 0.000 }
gfCNCPoint1[5234] = {X 155.8614, Y 48.9505, Z -1.3333, A 0.000, B 0.000, C 0.000 }
gfCNCPoint1[5235] = {X 157.1854, Y 48.5533, Z -1.3333, A 0.000, B 0.000, C 0.000 }
gfCNCPoint1[5236] = {X 158.2353, Y 48.3785, Z -1.3333, A 0.000, B 0.000, C 0.000 }
gfCNCPoint1[5237] = {X 159.2980, Y 48.3200, Z -1.3333, A 0.000, B 0.000, C 0.000 }
gfCNCPoint1[5238] = {X 176.3122, Y 48.3200, Z -1.3333, A 0.000, B 0.000, C 0.000 }
gfCNCPoint1[5239] = {X 175.1969, Y 47.6603, Z -1.3333, A 0.000, B 0.000, C 0.000 }
gfCNCPoint1[5240] = {X 174.1331, Y 46.9204, Z -1.3333, A 0.000, B 0.000, C 0.000 }
gfCNCPoint1[5241] = {X 172.7678, Y 45.7582, Z -1.3333, A 0.000, B 0.000, C 0.000 }
gfCNCPoint1[5242] = {X 171.5647, Y 44.4287, Z -1.3333, A 0.000, B 0.000, C 0.000 }
gfCNCPoint1[5243] = {X 170.6267, Y 43.0901, Z -1.3333, A 0.000, B 0.000, C 0.000 }
gfCNCPoint1[5244] = {X 169.8537, Y 41.6499, Z -1.3333, A 0.000, B 0.000, C 0.000 }
gfCNCPoint1[5245] = {X 169.2564, Y 40.1283, Z -1.3333, A 0.000, B 0.000, C 0.000 }
gfCNCPoint1[5246] = {X 168.8434, Y 38.5468, Z -1.3333, A 0.000, B 0.000, C 0.000 }
gfCNCPoint1[5247] = {X 168.6203, Y 36.9276, Z -1.3333, A 0.000, B 0.000, C 0.000 }
gfCNCPoint1[5248] = {X 168.5338, Y 35.0262, Z -1.3333, A 0.000, B 0.000, C 0.000 }
gfCNCPoint1[5249] = {X 168.6857, Y 33.1289, Z -1.3333, A 0.000, B 0.000, C 0.000 }
gfCNCPoint1[5250] = {X 169.0738, Y 31.2656, Z -1.3333, A 0.000, B 0.000, C 0.000 }
gfCNCPoint1[5251] = {X 169.6918, Y 29.4654, Z -1.3333, A 0.000, B 0.000, C 0.000 }
gfCNCPoint1[5252] = {X 170.2640, Y 28.2686, Z -1.3333, A 0.000, B 0.000, C 0.000 }
gfCNCPoint1[5253] = {X 170.9712, Y 27.1462, Z -1.3333, A 0.000, B 0.000, C 0.000 }
gfCNCPoint1[5254] = {X 171.8036, Y 26.1133, Z -1.3333, A 0.000, B 0.000, C 0.000 }
gfCNCPoint1[5255] = {X 172.7501, Y 25.1839, Z -1.3333, A 0.000, B 0.000, C 0.000 }
gfCNCPoint1[5256] = {X 173.7980, Y 24.3704, Z -1.3333, A 0.000, B 0.000, C 0.000 }
gfCNCPoint1[5257] = {X 173.0275, Y 23.7522, Z -1.3333, A 0.000, B 0.000, C 0.000 }
gfCNCPoint1[5258] = {X 172.3973, Y 22.9913, Z -1.3333, A 0.000, B 0.000, C 0.000 }
gfCNCPoint1[5259] = {X 171.9332, Y 22.1192, Z -1.3333, A 0.000, B 0.000, C 0.000 }
gfCNCPoint1[5260] = {X 169.3220, Y 15.7237, Z -1.3333, A 0.000, B 0.000, C 0.000 }
gfCNCPoint1[5261] = {X 169.1088, Y 15.0753, Z -1.3333, A 0.000, B 0.000, C 0.000 }
gfCNCPoint1[5262] = {X 168.9882, Y 14.4035, Z -1.3333, A 0.000, B 0.000, C 0.000 }
gfCNCPoint1[5263] = {X 168.9599, Y 13.8791, Z -1.3333, A 0.000, B 0.000, C 0.000 }
gfCNCPoint1[5264] = {X 168.9882, Y 13.3548, Z -1.3333, A 0.000, B 0.000, C 0.000 }
gfCNCPoint1[5265] = {X 169.1590, Y 12.4995, Z -1.3333, A 0.000, B 0.000, C 0.000 }
gfCNCPoint1[5266] = {X 169.4793, Y 11.6883, Z -1.3333, A 0.000, B 0.000, C 0.000 }
gfCNCPoint1[5267] = {X 169.9390, Y 10.9471, Z -1.3333, A 0.000, B 0.000, C 0.000 }
gfCNCPoint1[5268] = {X 170.6134, Y 10.2180, Z -1.3333, A 0.000, B 0.000, C 0.000 }
gfCNCPoint1[5269] = {X 171.4215, Y 9.6405, Z -1.3333, A 0.000, B 0.000, C 0.000 }
gfCNCPoint1[5270] = {X 172.0576, Y 9.2779, Z -1.3333, A 0.000, B 0.000, C 0.000 }
gfCNCPoint1[5271] = {X 172.9937, Y 8.8768, Z -1.3333, A 0.000, B 0.000, C 0.000 }
gfCNCPoint1[5272] = {X 173.9927, Y 8.6787, Z -1.3333, A 0.000, B 0.000, C 0.000 }
gfCNCPoint1[5273] = {X 175.0111, Y 8.6923, Z -1.3333, A 0.000, B 0.000, C 0.000 }
gfCNCPoint1[5274] = {X 176.0045, Y 8.9170, Z -1.3333, A 0.000, B 0.000, C 0.000 }
gfCNCPoint1[5275] = {X 177.7794, Y 8.1690, Z -1.3333, A 0.000, B 0.000, C 0.000 }
gfCNCPoint1[5276] = {X 179.6079, Y 7.5638, Z -1.3333, A 0.000, B 0.000, C 0.000 }
gfCNCPoint1[5277] = {X 181.4785, Y 7.1051, Z -1.3333, A 0.000, B 0.000, C 0.000 }
gfCNCPoint1[5278] = {X 168.0205, Y 7.1051, Z -1.3333, A 0.000, B 0.000, C 0.000 }
gfCNCPoint1[5279] = {X 168.0205, Y 4.7051, Z -1.3333, A 0.000, B 0.000, C 0.000 }
gfCNCPoint1[5280] = {X 155.1589, Y 4.7051, Z -1.3333, A 0.000, B 0.000, C 0.000 }
gfCNCPoint1[5281] = {X 155.1589, Y 7.1051, Z -1.3333, A 0.000, B 0.000, C 0.000 }
gfCNCPoint1[5282] = {X 137.3638, Y 7.1051, Z -1.3333, A 0.000, B 0.000, C 0.000 }
gfCNCPoint1[5283] = {X 137.5341, Y 7.2921, Z -1.3333, A 0.000, B 0.000, C 0.000 }
gfCNCPoint1[5284] = {X 137.6945, Y 7.4877, Z -1.3333, A 0.000, B 0.000, C 0.000 }
gfCNCPoint1[5285] = {X 154.8282, Y 7.4877, Z -1.3333, A 0.000, B 0.000, C 0.000 }
gfCNCPoint1[5286] = {X 154.9886, Y 7.2921, Z -1.3333, A 0.000, B 0.000, C 0.000 }
gfCNCPoint1[5287] = {X 155.1589, Y 7.1051, Z -1.3333, A 0.000, B 0.000, C 0.000 }
gfCNCPoint1[5288] = {X 155.1589, Y 4.7051, Z -1.3333, A 0.000, B 0.000, C 0.000 }
gfCNCPoint1[5289] = {X 23.8322, Y 4.7051, Z -1.3333, A 0.000, B 0.000, C 0.000 }
gfCNCPoint1[5290] = {X 25.7620, Y 5.7856, Z -1.3333, A 0.000, B 0.000, C 0.000 }
gfCNCPoint1[5291] = {X 27.5756, Y 7.0516, Z -1.3333, A 0.000, B 0.000, C 0.000 }
gfCNCPoint1[5292] = {X 28.5577, Y 7.8755, Z -1.3333, A 0.000, B 0.000, C 0.000 }
gfCNCPoint1[5293] = {X 29.4782, Y 8.7677, Z -1.3333, A 0.000, B 0.000, C 0.000 }
gfCNCPoint1[5294] = {X 30.6864, Y 10.1628, Z -1.3333, A 0.000, B 0.000, C 0.000 }
gfCNCPoint1[5295] = {X 31.7444, Y 11.6751, Z -1.3333, A 0.000, B 0.000, C 0.000 }
gfCNCPoint1[5296] = {X 32.6410, Y 13.2882, Z -1.3333, A 0.000, B 0.000, C 0.000 }
gfCNCPoint1[5297] = {X 33.3667, Y 14.9851, Z -1.3333, A 0.000, B 0.000, C 0.000 }
gfCNCPoint1[5298] = {X 33.9163, Y 16.8160, Z -1.3333, A 0.000, B 0.000, C 0.000 }
gfCNCPoint1[5299] = {X 34.2877, Y 18.6912, Z -1.3333, A 0.000, B 0.000, C 0.000 }
gfCNCPoint1[5300] = {X 34.4775, Y 20.5933, Z -1.3333, A 0.000, B 0.000, C 0.000 }
gfCNCPoint1[5301] = {X 34.4840, Y 22.5049, Z -1.3333, A 0.000, B 0.000, C 0.000 }
gfCNCPoint1[5302] = {X 34.3072, Y 24.4083, Z -1.3333, A 0.000, B 0.000, C 0.000 }
gfCNCPoint1[5303] = {X 33.9486, Y 26.2859, Z -1.3333, A 0.000, B 0.000, C 0.000 }
gfCNCPoint1[5304] = {X 33.4651, Y 27.9379, Z -1.3333, A 0.000, B 0.000, C 0.000 }
gfCNCPoint1[5305] = {X 32.8128, Y 29.5309, Z -1.3333, A 0.000, B 0.000, C 0.000 }
gfCNCPoint1[5306] = {X 31.9988, Y 31.0476, Z -1.3333, A 0.000, B 0.000, C 0.000 }
gfCNCPoint1[5307] = {X 32.1285, Y 31.2838, Z -1.3333, A 0.000, B 0.000, C 0.000 }
gfCNCPoint1[5308] = {X 32.2513, Y 31.5237, Z -1.3333, A 0.000, B 0.000, C 0.000 }
gfCNCPoint1[5309] = {X 35.3025, Y 37.8269, Z -1.3333, A 0.000, B 0.000, C 0.000 }
gfCNCPoint1[5310] = {X 35.7263, Y 38.8573, Z -1.3333, A 0.000, B 0.000, C 0.000 }
gfCNCPoint1[5311] = {X 36.0224, Y 39.9313, Z -1.3333, A 0.000, B 0.000, C 0.000 }
gfCNCPoint1[5312] = {X 36.1865, Y 41.0332, Z -1.3333, A 0.000, B 0.000, C 0.000 }
gfCNCPoint1[5313] = {X 36.2163, Y 42.1469, Z -1.3333, A 0.000, B 0.000, C 0.000 }
gfCNCPoint1[5314] = {X 36.6306, Y 41.4258, Z -1.3333, A 0.000, B 0.000, C 0.000 }
gfCNCPoint1[5315] = {X 37.1614, Y 40.7855, Z -1.3333, A 0.000, B 0.000, C 0.000 }
gfCNCPoint1[5316] = {X 37.7932, Y 40.2447, Z -1.3333, A 0.000, B 0.000, C 0.000 }
gfCNCPoint1[5317] = {X 38.5077, Y 39.8189, Z -1.3333, A 0.000, B 0.000, C 0.000 }
gfCNCPoint1[5318] = {X 39.0460, Y 38.5335, Z -1.3333, A 0.000, B 0.000, C 0.000 }
gfCNCPoint1[5319] = {X 39.5419, Y 37.2312, Z -1.3333, A 0.000, B 0.000, C 0.000 }
gfCNCPoint1[5320] = {X 47.6703, Y 15.4045, Z -1.3333, A 0.000, B 0.000, C 0.000 }
gfCNCPoint1[5321] = {X 47.3200, Y 14.6512, Z -1.3333, A 0.000, B 0.000, C 0.000 }
gfCNCPoint1[5322] = {X 47.1026, Y 13.8493, Z -1.3333, A 0.000, B 0.000, C 0.000 }
gfCNCPoint1[5323] = {X 47.0244, Y 13.0222, Z -1.3333, A 0.000, B 0.000, C 0.000 }
gfCNCPoint1[5324] = {X 47.0242, Y 12.1868, Z -1.3333, A 0.000, B 0.000, C 0.000 }
gfCNCPoint1[5325] = {X 47.0722, Y 11.5041, Z -1.3333, A 0.000, B 0.000, C 0.000 }
gfCNCPoint1[5326] = {X 47.2152, Y 10.8349, Z -1.3333, A 0.000, B 0.000, C 0.000 }
gfCNCPoint1[5327] = {X 42.6031, Y 9.5051, Z -1.3333, A 0.000, B 0.000, C 0.000 }
gfCNCPoint1[5328] = {X 36.0437, Y 9.5051, Z -1.3333, A 0.000, B 0.000, C 0.000 }
gfCNCPoint1[5329] = {X 37.0537, Y 11.3877, Z -1.3333, A 0.000, B 0.000, C 0.000 }
gfCNCPoint1[5330] = {X 37.8822, Y 13.3569, Z -1.3333, A 0.000, B 0.000, C 0.000 }
gfCNCPoint1[5331] = {X 38.5451, Y 15.5408, Z -1.3333, A 0.000, B 0.000, C 0.000 }
gfCNCPoint1[5332] = {X 39.0036, Y 17.7766, Z -1.3333, A 0.000, B 0.000, C 0.000 }
gfCNCPoint1[5333] = {X 39.2538, Y 20.0451, Z -1.3333, A 0.000, B 0.000, C 0.000 }
gfCNCPoint1[5334] = {X 39.2937, Y 22.3271, Z -1.3333, A 0.000, B 0.000, C 0.000 }
gfCNCPoint1[5335] = {X 39.1227, Y 24.6030, Z -1.3333, A 0.000, B 0.000, C 0.000 }
gfCNCPoint1[5336] = {X 42.5394, Y 15.4282, Z -1.3333, A 0.000, B 0.000, C 0.000 }
gfCNCPoint1[5337] = {X 42.3075, Y 14.2453, Z -1.3333, A 0.000, B 0.000, C 0.000 }
gfCNCPoint1[5338] = {X 42.2244, Y 13.0428, Z -1.3333, A 0.000, B 0.000, C 0.000 }
gfCNCPoint1[5339] = {X 42.2242, Y 12.1868, Z -1.3333, A 0.000, B 0.000, C 0.000 }
gfCNCPoint1[5340] = {X 42.3194, Y 10.8326, Z -1.3333, A 0.000, B 0.000, C 0.000 }
gfCNCPoint1[5341] = {X 42.6031, Y 9.5051, Z -1.3333, A 0.000, B 0.000, C 0.000 }
gfCNCPoint1[5342] = {X 44.9092, Y 10.1700, Z -1.3333, A 0.000, B 0.000, C 0.000 }
gfCNCPoint1[5343] = {X 45.3322, Y 9.0551, Z -1.3333, A 0.000, B 0.000, C 0.000 }
gfCNCPoint1[5344] = {X 45.9316, Y 8.0243, Z -1.3333, A 0.000, B 0.000, C 0.000 }
gfCNCPoint1[5345] = {X 46.6913, Y 7.1051, Z -1.3333, A 0.000, B 0.000, C 0.000 }
gfCNCPoint1[5346] = {X 31.2091, Y 7.1051, Z -1.3333, A 0.000, B 0.000, C 0.000 }
gfCNCPoint1[5347] = {X 32.2246, Y 8.2453, Z -1.3333, A 0.000, B 0.000, C 0.000 }
gfCNCPoint1[5348] = {X 33.1515, Y 9.4585, Z -1.3333, A 0.000, B 0.000, C 0.000 }
gfCNCPoint1[5349] = {X 33.9846, Y 10.7380, Z -1.3333, A 0.000, B 0.000, C 0.000 }
gfCNCPoint1[5350] = {X 34.8851, Y 12.4160, Z -1.3333, A 0.000, B 0.000, C 0.000 }
gfCNCPoint1[5351] = {X 35.6245, Y 14.1710, Z -1.3333, A 0.000, B 0.000, C 0.000 }
gfCNCPoint1[5352] = {X 36.2212, Y 16.1407, Z -1.3333, A 0.000, B 0.000, C 0.000 }
gfCNCPoint1[5353] = {X 36.6339, Y 18.1570, Z -1.3333, A 0.000, B 0.000, C 0.000 }
gfCNCPoint1[5354] = {X 36.8590, Y 20.2028, Z -1.3333, A 0.000, B 0.000, C 0.000 }
gfCNCPoint1[5355] = {X 36.8946, Y 22.2606, Z -1.3333, A 0.000, B 0.000, C 0.000 }
gfCNCPoint1[5356] = {X 36.7403, Y 24.3129, Z -1.3333, A 0.000, B 0.000, C 0.000 }
gfCNCPoint1[5357] = {X 36.5481, Y 25.5851, Z -1.3333, A 0.000, B 0.000, C 0.000 }
gfCNCPoint1[5358] = {X 36.2827, Y 26.8441, Z -1.3333, A 0.000, B 0.000, C 0.000 }
gfCNCPoint1[5359] = {X 35.8740, Y 28.3041, Z -1.3333, A 0.000, B 0.000, C 0.000 }
gfCNCPoint1[5360] = {X 35.3500, Y 29.7268, Z -1.3333, A 0.000, B 0.000, C 0.000 }
gfCNCPoint1[5361] = {X 34.7141, Y 31.1031, Z -1.3333, A 0.000, B 0.000, C 0.000 }
gfCNCPoint1[5362] = {X 37.2852, Y 36.4144, Z -1.3333, A 0.000, B 0.000, C 0.000 }
gfCNCPoint1[5363] = {X 45.0744, Y 15.4982, Z -1.3333, A 0.000, B 0.000, C 0.000 }
gfCNCPoint1[5364] = {X 44.7426, Y 14.2853, Z -1.3333, A 0.000, B 0.000, C 0.000 }
gfCNCPoint1[5365] = {X 44.6244, Y 13.0334, Z -1.3333, A 0.000, B 0.000, C 0.000 }
gfCNCPoint1[5366] = {X 44.6242, Y 12.1868, Z -1.3333, A 0.000, B 0.000, C 0.000 }
gfCNCPoint1[5367] = {X 44.6958, Y 11.1684, Z -1.3333, A 0.000, B 0.000, C 0.000 }
gfCNCPoint1[5368] = {X 44.9092, Y 10.1700, Z -1.3333, A 0.000, B 0.000, C 0.000 }
gfCNCPoint1[5369] = {X 47.2152, Y 10.8349, Z -1.3333, A 0.000, B 0.000, C 0.000 }
gfCNCPoint1[5370] = {X 47.4988, Y 10.0876, Z -1.3333, A 0.000, B 0.000, C 0.000 }
gfCNCPoint1[5371] = {X 47.9006, Y 9.3965, Z -1.3333, A 0.000, B 0.000, C 0.000 }
gfCNCPoint1[5372] = {X 48.4098, Y 8.7804, Z -1.3333, A 0.000, B 0.000, C 0.000 }
gfCNCPoint1[5373] = {X 49.1544, Y 8.1553, Z -1.3333, A 0.000, B 0.000, C 0.000 }
gfCNCPoint1[5374] = {X 50.0080, Y 7.6903, Z -1.3333, A 0.000, B 0.000, C 0.000 }
gfCNCPoint1[5375] = {X 50.9369, Y 7.4036, Z -1.3333, A 0.000, B 0.000, C 0.000 }
gfCNCPoint1[5376] = {X 51.9042, Y 7.3068, Z -1.3333, A 0.000, B 0.000, C 0.000 }
gfCNCPoint1[5377] = {X 59.6221, Y 7.3068, Z -1.3333, A 0.000, B 0.000, C 0.000 }
gfCNCPoint1[5378] = {X 60.5894, Y 7.4036, Z -1.3333, A 0.000, B 0.000, C 0.000 }
gfCNCPoint1[5379] = {X 61.5183, Y 7.6903, Z -1.3333, A 0.000, B 0.000, C 0.000 }
gfCNCPoint1[5380] = {X 62.3720, Y 8.1553, Z -1.3333, A 0.000, B 0.000, C 0.000 }
gfCNCPoint1[5381] = {X 63.1165, Y 8.7804, Z -1.3333, A 0.000, B 0.000, C 0.000 }
gfCNCPoint1[5382] = {X 63.7054, Y 9.5145, Z -1.3333, A 0.000, B 0.000, C 0.000 }
gfCNCPoint1[5383] = {X 64.1425, Y 10.3481, Z -1.3333, A 0.000, B 0.000, C 0.000 }
gfCNCPoint1[5384] = {X 64.4114, Y 11.2500, Z -1.3333, A 0.000, B 0.000, C 0.000 }
gfCNCPoint1[5385] = {X 64.5021, Y 12.1868, Z -1.3333, A 0.000, B 0.000, C 0.000 }
gfCNCPoint1[5386] = {X 64.5019, Y 13.0237, Z -1.3333, A 0.000, B 0.000, C 0.000 }
gfCNCPoint1[5387] = {X 64.4204, Y 13.8672, Z -1.3333, A 0.000, B 0.000, C 0.000 }
gfCNCPoint1[5388] = {X 64.1942, Y 14.6839, Z -1.3333, A 0.000, B 0.000, C 0.000 }
gfCNCPoint1[5389] = {X 63.8302, Y 15.4492, Z -1.3333, A 0.000, B 0.000, C 0.000 }
gfCNCPoint1[5390] = {X 63.9941, Y 15.8774, Z -1.3333, A 0.000, B 0.000, C 0.000 }
gfCNCPoint1[5391] = {X 72.9528, Y 39.8570, Z -1.3333, A 0.000, B 0.000, C 0.000 }
gfCNCPoint1[5392] = {X 73.8432, Y 40.4389, Z -1.3333, A 0.000, B 0.000, C 0.000 }
gfCNCPoint1[5393] = {X 74.5864, Y 41.1999, Z -1.3333, A 0.000, B 0.000, C 0.000 }
gfCNCPoint1[5394] = {X 75.1471, Y 42.1038, Z -1.3333, A 0.000, B 0.000, C 0.000 }
gfCNCPoint1[5395] = {X 75.4986, Y 43.1078, Z -1.3333, A 0.000, B 0.000, C 0.000 }
gfCNCPoint1[5396] = {X 75.6243, Y 44.1640, Z -1.3333, A 0.000, B 0.000, C 0.000 }
gfCNCPoint1[5397] = {X 75.6245, Y 45.0000, Z -1.3333, A 0.000, B 0.000, C 0.000 }
gfCNCPoint1[5398] = {X 75.5307, Y 45.9520, Z -1.3333, A 0.000, B 0.000, C 0.000 }
gfCNCPoint1[5399] = {X 75.2530, Y 46.8675, Z -1.3333, A 0.000, B 0.000, C 0.000 }
gfCNCPoint1[5400] = {X 74.8020, Y 47.7112, Z -1.3333, A 0.000, B 0.000, C 0.000 }
gfCNCPoint1[5401] = {X 74.1951, Y 48.4507, Z -1.3333, A 0.000, B 0.000, C 0.000 }
gfCNCPoint1[5402] = {X 73.4556, Y 49.0576, Z -1.3333, A 0.000, B 0.000, C 0.000 }
gfCNCPoint1[5403] = {X 72.6120, Y 49.5085, Z -1.3333, A 0.000, B 0.000, C 0.000 }
gfCNCPoint1[5404] = {X 71.6965, Y 49.7862, Z -1.3333, A 0.000, B 0.000, C 0.000 }
gfCNCPoint1[5405] = {X 70.7445, Y 49.8800, Z -1.3333, A 0.000, B 0.000, C 0.000 }
gfCNCPoint1[5406] = {X 64.1851, Y 49.8800, Z -1.3333, A 0.000, B 0.000, C 0.000 }
gfCNCPoint1[5407] = {X 63.2331, Y 49.7862, Z -1.3333, A 0.000, B 0.000, C 0.000 }
gfCNCPoint1[5408] = {X 62.3176, Y 49.5085, Z -1.3333, A 0.000, B 0.000, C 0.000 }
gfCNCPoint1[5409] = {X 61.4740, Y 49.0576, Z -1.3333, A 0.000, B 0.000, C 0.000 }
gfCNCPoint1[5410] = {X 60.7345, Y 48.4507, Z -1.3333, A 0.000, B 0.000, C 0.000 }
gfCNCPoint1[5411] = {X 60.1276, Y 47.7112, Z -1.3333, A 0.000, B 0.000, C 0.000 }
gfCNCPoint1[5412] = {X 59.6766, Y 46.8675, Z -1.3333, A 0.000, B 0.000, C 0.000 }
gfCNCPoint1[5413] = {X 59.3989, Y 45.9520, Z -1.3333, A 0.000, B 0.000, C 0.000 }
gfCNCPoint1[5414] = {X 59.3051, Y 45.0000, Z -1.3333, A 0.000, B 0.000, C 0.000 }
gfCNCPoint1[5415] = {X 59.3052, Y 44.2029, Z -1.3333, A 0.000, B 0.000, C 0.000 }
gfCNCPoint1[5416] = {X 59.3848, Y 43.3307, Z -1.3333, A 0.000, B 0.000, C 0.000 }
gfCNCPoint1[5417] = {X 59.6191, Y 42.4868, Z -1.3333, A 0.000, B 0.000, C 0.000 }
gfCNCPoint1[5418] = {X 60.0004, Y 41.6983, Z -1.3333, A 0.000, B 0.000, C 0.000 }
gfCNCPoint1[5419] = {X 59.6162, Y 40.6492, Z -1.3333, A 0.000, B 0.000, C 0.000 }
gfCNCPoint1[5420] = {X 52.4652, Y 40.6492, Z -1.3333, A 0.000, B 0.000, C 0.000 }
gfCNCPoint1[5421] = {X 51.9462, Y 42.0434, Z -1.3333, A 0.000, B 0.000, C 0.000 }
gfCNCPoint1[5422] = {X 52.2213, Y 42.7232, Z -1.3333, A 0.000, B 0.000, C 0.000 }
gfCNCPoint1[5423] = {X 52.3914, Y 43.4365, Z -1.3333, A 0.000, B 0.000, C 0.000 }
gfCNCPoint1[5424] = {X 52.4528, Y 44.1672, Z -1.3333, A 0.000, B 0.000, C 0.000 }
gfCNCPoint1[5425] = {X 52.4529, Y 45.0000, Z -1.3333, A 0.000, B 0.000, C 0.000 }
gfCNCPoint1[5426] = {X 52.3592, Y 45.9520, Z -1.3333, A 0.000, B 0.000, C 0.000 }
gfCNCPoint1[5427] = {X 52.0815, Y 46.8675, Z -1.3333, A 0.000, B 0.000, C 0.000 }
gfCNCPoint1[5428] = {X 51.6305, Y 47.7112, Z -1.3333, A 0.000, B 0.000, C 0.000 }
gfCNCPoint1[5429] = {X 51.0236, Y 48.4507, Z -1.3333, A 0.000, B 0.000, C 0.000 }
gfCNCPoint1[5430] = {X 50.2841, Y 49.0576, Z -1.3333, A 0.000, B 0.000, C 0.000 }
gfCNCPoint1[5431] = {X 49.4404, Y 49.5085, Z -1.3333, A 0.000, B 0.000, C 0.000 }
gfCNCPoint1[5432] = {X 48.5250, Y 49.7862, Z -1.3333, A 0.000, B 0.000, C 0.000 }
gfCNCPoint1[5433] = {X 47.5729, Y 49.8800, Z -1.3333, A 0.000, B 0.000, C 0.000 }
gfCNCPoint1[5434] = {X 40.6393, Y 49.8800, Z -1.3333, A 0.000, B 0.000, C 0.000 }
gfCNCPoint1[5435] = {X 39.6433, Y 49.7773, Z -1.3333, A 0.000, B 0.000, C 0.000 }
gfCNCPoint1[5436] = {X 38.6892, Y 49.4734, Z -1.3333, A 0.000, B 0.000, C 0.000 }
gfCNCPoint1[5437] = {X 37.8173, Y 48.9813, Z -1.3333, A 0.000, B 0.000, C 0.000 }
gfCNCPoint1[5438] = {X 37.0641, Y 48.3215, Z -1.3333, A 0.000, B 0.000, C 0.000 }
gfCNCPoint1[5439] = {X 36.5085, Y 47.5983, Z -1.3333, A 0.000, B 0.000, C 0.000 }
gfCNCPoint1[5440] = {X 36.0972, Y 46.7843, Z -1.3333, A 0.000, B 0.000, C 0.000 }
gfCNCPoint1[5441] = {X 35.8445, Y 45.9080, Z -1.3333, A 0.000, B 0.000, C 0.000 }
gfCNCPoint1[5442] = {X 35.7593, Y 45.0000, Z -1.3333, A 0.000, B 0.000, C 0.000 }
gfCNCPoint1[5443] = {X 35.7593, Y 44.7148, Z -1.3333, A 0.000, B 0.000, C 0.000 }
gfCNCPoint1[5444] = {X 36.2393, Y 44.7148, Z -1.3333, A 0.000, B 0.000, C 0.000 }
gfCNCPoint1[5445] = {X 36.2397, Y 44.1483, Z -1.3333, A 0.000, B 0.000, C 0.000 }
gfCNCPoint1[5446] = {X 36.3681, Y 43.1518, Z -1.3333, A 0.000, B 0.000, C 0.000 }
gfCNCPoint1[5447] = {X 36.7192, Y 42.2105, Z -1.3333, A 0.000, B 0.000, C 0.000 }
gfCNCPoint1[5448] = {X 37.2747, Y 41.3734, Z -1.3333, A 0.000, B 0.000, C 0.000 }
gfCNCPoint1[5449] = {X 38.0056, Y 40.6841, Z -1.3333, A 0.000, B 0.000, C 0.000 }
gfCNCPoint1[5450] = {X 38.8738, Y 40.1785, Z -1.3333, A 0.000, B 0.000, C 0.000 }
gfCNCPoint1[5451] = {X 39.4569, Y 38.7983, Z -1.3333, A 0.000, B 0.000, C 0.000 }
gfCNCPoint1[5452] = {X 39.9917, Y 37.3987, Z -1.3333, A 0.000, B 0.000, C 0.000 }
gfCNCPoint1[5453] = {X 48.2011, Y 15.3544, Z -1.3333, A 0.000, B 0.000, C 0.000 }
gfCNCPoint1[5454] = {X 47.8187, Y 14.6115, Z -1.3333, A 0.000, B 0.000, C 0.000 }
gfCNCPoint1[5455] = {X 47.5835, Y 13.8097, Z -1.3333, A 0.000, B 0.000, C 0.000 }
gfCNCPoint1[5456] = {X 47.5042, Y 12.9779, Z -1.3333, A 0.000, B 0.000, C 0.000 }
gfCNCPoint1[5457] = {X 47.5042, Y 12.1868, Z -1.3333, A 0.000, B 0.000, C 0.000 }
gfCNCPoint1[5458] = {X 47.6145, Y 11.2077, Z -1.3333, A 0.000, B 0.000, C 0.000 }
gfCNCPoint1[5459] = {X 47.9400, Y 10.2777, Z -1.3333, A 0.000, B 0.000, C 0.000 }
gfCNCPoint1[5460] = {X 48.4642, Y 9.4435, Z -1.3333, A 0.000, B 0.000, C 0.000 }
gfCNCPoint1[5461] = {X 49.1609, Y 8.7468, Z -1.3333, A 0.000, B 0.000, C 0.000 }
gfCNCPoint1[5462] = {X 49.9951, Y 8.2226, Z -1.3333, A 0.000, B 0.000, C 0.000 }
gfCNCPoint1[5463] = {X 50.9251, Y 7.8971, Z -1.3333, A 0.000, B 0.000, C 0.000 }
gfCNCPoint1[5464] = {X 51.9042, Y 7.7868, Z -1.3333, A 0.000, B 0.000, C 0.000 }
gfCNCPoint1[5465] = {X 59.6221, Y 7.7868, Z -1.3333, A 0.000, B 0.000, C 0.000 }
gfCNCPoint1[5466] = {X 60.6012, Y 7.8971, Z -1.3333, A 0.000, B 0.000, C 0.000 }
gfCNCPoint1[5467] = {X 61.5312, Y 8.2226, Z -1.3333, A 0.000, B 0.000, C 0.000 }
gfCNCPoint1[5468] = {X 62.3655, Y 8.7468, Z -1.3333, A 0.000, B 0.000, C 0.000 }
gfCNCPoint1[5469] = {X 63.0622, Y 9.4435, Z -1.3333, A 0.000, B 0.000, C 0.000 }
gfCNCPoint1[5470] = {X 63.5864, Y 10.2777, Z -1.3333, A 0.000, B 0.000, C 0.000 }
gfCNCPoint1[5471] = {X 63.9118, Y 11.2077, Z -1.3333, A 0.000, B 0.000, C 0.000 }
gfCNCPoint1[5472] = {X 64.0221, Y 12.1868, Z -1.3333, A 0.000, B 0.000, C 0.000 }
gfCNCPoint1[5473] = {X 64.0219, Y 13.0233, Z -1.3333, A 0.000, B 0.000, C 0.000 }
gfCNCPoint1[5474] = {X 63.9335, Y 13.8565, Z -1.3333, A 0.000, B 0.000, C 0.000 }
gfCNCPoint1[5475] = {X 63.6888, Y 14.6578, Z -1.3333, A 0.000, B 0.000, C 0.000 }
gfCNCPoint1[5476] = {X 63.2967, Y 15.3983, Z -1.3333, A 0.000, B 0.000, C 0.000 }
gfCNCPoint1[5477] = {X 63.5448, Y 16.0465, Z -1.3333, A 0.000, B 0.000, C 0.000 }
gfCNCPoint1[5478] = {X 66.1090, Y 22.8602, Z -1.3333, A 0.000, B 0.000, C 0.000 }
gfCNCPoint1[5479] = {X 72.2830, Y 39.4717, Z -1.3333, A 0.000, B 0.000, C 0.000 }
gfCNCPoint1[5480] = {X 72.5758, Y 40.2080, Z -1.3333, A 0.000, B 0.000, C 0.000 }
gfCNCPoint1[5481] = {X 73.4338, Y 40.7263, Z -1.3333, A 0.000, B 0.000, C 0.000 }
gfCNCPoint1[5482] = {X 74.1522, Y 41.4254, Z -1.3333, A 0.000, B 0.000, C 0.000 }
gfCNCPoint1[5483] = {X 74.6937, Y 42.2689, Z -1.3333, A 0.000, B 0.000, C 0.000 }
gfCNCPoint1[5484] = {X 75.0303, Y 43.2131, Z -1.3333, A 0.000, B 0.000, C 0.000 }
gfCNCPoint1[5485] = {X 75.1445, Y 44.2089, Z -1.3333, A 0.000, B 0.000, C 0.000 }
gfCNCPoint1[5486] = {X 75.1445, Y 45.0000, Z -1.3333, A 0.000, B 0.000, C 0.000 }
gfCNCPoint1[5487] = {X 75.0341, Y 45.9791, Z -1.3333, A 0.000, B 0.000, C 0.000 }
gfCNCPoint1[5488] = {X 74.7087, Y 46.9091, Z -1.3333, A 0.000, B 0.000, C 0.000 }
gfCNCPoint1[5489] = {X 74.1845, Y 47.7434, Z -1.3333, A 0.000, B 0.000, C 0.000 }
gfCNCPoint1[5490] = {X 73.4878, Y 48.4401, Z -1.3333, A 0.000, B 0.000, C 0.000 }
gfCNCPoint1[5491] = {X 72.6535, Y 48.9643, Z -1.3333, A 0.000, B 0.000, C 0.000 }
gfCNCPoint1[5492] = {X 71.7236, Y 49.2897, Z -1.3333, A 0.000, B 0.000, C 0.000 }
gfCNCPoint1[5493] = {X 70.7445, Y 49.4000, Z -1.3333, A 0.000, B 0.000, C 0.000 }
gfCNCPoint1[5494] = {X 64.1851, Y 49.4000, Z -1.3333, A 0.000, B 0.000, C 0.000 }
gfCNCPoint1[5495] = {X 63.2060, Y 49.2897, Z -1.3333, A 0.000, B 0.000, C 0.000 }
gfCNCPoint1[5496] = {X 62.2760, Y 48.9643, Z -1.3333, A 0.000, B 0.000, C 0.000 }
gfCNCPoint1[5497] = {X 61.4418, Y 48.4401, Z -1.3333, A 0.000, B 0.000, C 0.000 }
gfCNCPoint1[5498] = {X 60.7451, Y 47.7434, Z -1.3333, A 0.000, B 0.000, C 0.000 }
gfCNCPoint1[5499] = {X 60.2209, Y 46.9091, Z -1.3333, A 0.000, B 0.000, C 0.000 }
gfCNCPoint1[5500] = {X 59.8955, Y 45.9791, Z -1.3333, A 0.000, B 0.000, C 0.000 }
gfCNCPoint1[5501] = {X 59.7851, Y 45.0000, Z -1.3333, A 0.000, B 0.000, C 0.000 }
gfCNCPoint1[5502] = {X 59.7856, Y 44.1483, Z -1.3333, A 0.000, B 0.000, C 0.000 }
gfCNCPoint1[5503] = {X 59.8785, Y 43.3074, Z -1.3333, A 0.000, B 0.000, C 0.000 }
gfCNCPoint1[5504] = {X 60.1306, Y 42.4999, Z -1.3333, A 0.000, B 0.000, C 0.000 }
gfCNCPoint1[5505] = {X 60.5326, Y 41.7555, Z -1.3333, A 0.000, B 0.000, C 0.000 }
gfCNCPoint1[5506] = {X 59.9516, Y 40.1692, Z -1.3333, A 0.000, B 0.000, C 0.000 }
gfCNCPoint1[5507] = {X 52.1317, Y 40.1692, Z -1.3333, A 0.000, B 0.000, C 0.000 }
gfCNCPoint1[5508] = {X 51.4217, Y 42.0765, Z -1.3333, A 0.000, B 0.000, C 0.000 }
gfCNCPoint1[5509] = {X 51.7250, Y 42.7528, Z -1.3333, A 0.000, B 0.000, C 0.000 }
gfCNCPoint1[5510] = {X 51.9105, Y 43.4704, Z -1.3333, A 0.000, B 0.000, C 0.000 }
gfCNCPoint1[5511] = {X 51.9729, Y 44.2089, Z -1.3333, A 0.000, B 0.000, C 0.000 }
gfCNCPoint1[5512] = {X 51.9729, Y 45.0000, Z -1.3333, A 0.000, B 0.000, C 0.000 }
gfCNCPoint1[5513] = {X 51.8626, Y 45.9791, Z -1.3333, A 0.000, B 0.000, C 0.000 }
gfCNCPoint1[5514] = {X 51.5372, Y 46.9091, Z -1.3333, A 0.000, B 0.000, C 0.000 }
gfCNCPoint1[5515] = {X 51.0130, Y 47.7434, Z -1.3333, A 0.000, B 0.000, C 0.000 }
gfCNCPoint1[5516] = {X 50.3163, Y 48.4401, Z -1.3333, A 0.000, B 0.000, C 0.000 }
gfCNCPoint1[5517] = {X 49.4820, Y 48.9643, Z -1.3333, A 0.000, B 0.000, C 0.000 }
gfCNCPoint1[5518] = {X 48.5520, Y 49.2897, Z -1.3333, A 0.000, B 0.000, C 0.000 }
gfCNCPoint1[5519] = {X 47.5729, Y 49.4000, Z -1.3333, A 0.000, B 0.000, C 0.000 }
gfCNCPoint1[5520] = {X 40.6393, Y 49.4000, Z -1.3333, A 0.000, B 0.000, C 0.000 }
gfCNCPoint1[5521] = {X 39.6602, Y 49.2897, Z -1.3333, A 0.000, B 0.000, C 0.000 }
gfCNCPoint1[5522] = {X 38.7302, Y 48.9643, Z -1.3333, A 0.000, B 0.000, C 0.000 }
gfCNCPoint1[5523] = {X 37.8959, Y 48.4401, Z -1.3333, A 0.000, B 0.000, C 0.000 }
gfCNCPoint1[5524] = {X 37.1992, Y 47.7434, Z -1.3333, A 0.000, B 0.000, C 0.000 }
gfCNCPoint1[5525] = {X 36.6750, Y 46.9091, Z -1.3333, A 0.000, B 0.000, C 0.000 }
gfCNCPoint1[5526] = {X 36.3496, Y 45.9791, Z -1.3333, A 0.000, B 0.000, C 0.000 }
gfCNCPoint1[5527] = {X 36.2393, Y 45.0000, Z -1.3333, A 0.000, B 0.000, C 0.000 }
gfCNCPoint1[5528] = {X 36.2393, Y 44.7148, Z -1.3333, A 0.000, B 0.000, C 0.000 }
gfCNCPoint1[5529] = {X 35.7593, Y 44.7148, Z -1.3333, A 0.000, B 0.000, C 0.000 }
gfCNCPoint1[5530] = {X 35.2211, Y 46.0074, Z -1.3333, A 0.000, B 0.000, C 0.000 }
gfCNCPoint1[5531] = {X 34.4930, Y 47.2034, Z -1.3333, A 0.000, B 0.000, C 0.000 }
gfCNCPoint1[5532] = {X 33.5918, Y 48.2750, Z -1.3333, A 0.000, B 0.000, C 0.000 }
gfCNCPoint1[5533] = {X 33.2092, Y 48.6435, Z -1.3333, A 0.000, B 0.000, C 0.000 }
gfCNCPoint1[5534] = {X 32.8060, Y 48.9892, Z -1.3333, A 0.000, B 0.000, C 0.000 }
gfCNCPoint1[5535] = {X 32.2636, Y 49.4277, Z -1.3333, A 0.000, B 0.000, C 0.000 }
gfCNCPoint1[5536] = {X 31.1778, Y 50.1812, Z -1.3333, A 0.000, B 0.000, C 0.000 }
gfCNCPoint1[5537] = {X 29.9953, Y 50.7717, Z -1.3333, A 0.000, B 0.000, C 0.000 }
gfCNCPoint1[5538] = {X 28.7406, Y 51.1870, Z -1.3333, A 0.000, B 0.000, C 0.000 }
gfCNCPoint1[5539] = {X 27.4394, Y 51.4187, Z -1.3333, A 0.000, B 0.000, C 0.000 }
gfCNCPoint1[5540] = {X 26.1184, Y 51.4618, Z -1.3333, A 0.000, B 0.000, C 0.000 }
gfCNCPoint1[5541] = {X 24.2244, Y 52.3516, Z -1.3333, A 0.000, B 0.000, C 0.000 }
gfCNCPoint1[5542] = {X 22.2783, Y 53.1207, Z -1.3333, A 0.000, B 0.000, C 0.000 }
gfCNCPoint1[5543] = {X 20.2878, Y 53.7661, Z -1.3333, A 0.000, B 0.000, C 0.000 }
gfCNCPoint1[5544] = {X 19.7489, Y 53.9156, Z -1.3333, A 0.000, B 0.000, C 0.000 }
gfCNCPoint1[5545] = {X 17.4808, Y 54.4405, Z -1.3333, A 0.000, B 0.000, C 0.000 }
gfCNCPoint1[5546] = {X 15.1761, Y 54.7691, Z -1.3333, A 0.000, B 0.000, C 0.000 }
gfCNCPoint1[5547] = {X 12.8517, Y 54.8989, Z -1.3333, A 0.000, B 0.000, C 0.000 }
gfCNCPoint1[5548] = {X 10.5247, Y 54.8292, Z -1.3333, A 0.000, B 0.000, C 0.000 }
gfCNCPoint1[5549] = {X 8.2122, Y 54.5603, Z -1.3333, A 0.000, B 0.000, C 0.000 }
gfCNCPoint1[5550] = {X 7.8656, Y 54.5077, Z -1.3333, A 0.000, B 0.000, C 0.000 }
gfCNCPoint1[5551] = {X 7.5198, Y 54.4497, Z -1.3333, A 0.000, B 0.000, C 0.000 }
gfCNCPoint1[5552] = {X 6.1003, Y 54.1511, Z -1.3333, A 0.000, B 0.000, C 0.000 }
gfCNCPoint1[5553] = {X 4.7035, Y 53.7597, Z -1.3333, A 0.000, B 0.000, C 0.000 }
gfCNCPoint1[5554] = {X 4.7035, Y 95.2949, Z -1.3333, A 0.000, B 0.000, C 0.000 }
gfCNCPoint1[5555] = {X 117.9387, Y 95.2949, Z -1.3333, A 0.000, B 0.000, C 0.000 }
gfCNCPoint1[5556] = {X 118.3620, Y 94.0767, Z -1.3333, A 0.000, B 0.000, C 0.000 }
gfCNCPoint1[5557] = {X 118.9937, Y 92.9523, Z -1.3333, A 0.000, B 0.000, C 0.000 }
gfCNCPoint1[5558] = {X 119.8138, Y 91.9569, Z -1.3333, A 0.000, B 0.000, C 0.000 }
gfCNCPoint1[5559] = {X 120.7967, Y 91.1220, Z -1.3333, A 0.000, B 0.000, C 0.000 }
gfCNCPoint1[5560] = {X 121.9115, Y 90.4735, Z -1.3333, A 0.000, B 0.000, C 0.000 }
gfCNCPoint1[5561] = {X 123.1232, Y 90.0320, Z -1.3333, A 0.000, B 0.000, C 0.000 }
gfCNCPoint1[5562] = {X 124.3939, Y 89.8112, Z -1.3333, A 0.000, B 0.000, C 0.000 }
gfCNCPoint1[5563] = {X 125.0451, Y 89.7132, Z -1.3333, A 0.000, B 0.000, C 0.000 }
gfCNCPoint1[5564] = {X 125.3563, Y 89.6662, Z -1.3333, A 0.000, B 0.000, C 0.000 }
gfCNCPoint1[5565] = {X 125.6659, Y 89.6091, Z -1.3333, A 0.000, B 0.000, C 0.000 }
gfCNCPoint1[5566] = {X 126.4929, Y 88.7982, Z -1.3333, A 0.000, B 0.000, C 0.000 }
gfCNCPoint1[5567] = {X 127.2857, Y 87.9539, Z -1.3333, A 0.000, B 0.000, C 0.000 }
gfCNCPoint1[5568] = {X 152.2078, Y 60.5859, Z -1.3333, A 0.000, B 0.000, C 0.000 }
gfCNCPoint1[5569] = {X 152.0685, Y 59.7905, Z -1.3333, A 0.000, B 0.000, C 0.000 }
gfCNCPoint1[5570] = {X 152.0181, Y 58.9845, Z -1.3333, A 0.000, B 0.000, C 0.000 }
gfCNCPoint1[5571] = {X 152.0180, Y 58.0000, Z -1.3333, A 0.000, B 0.000, C 0.000 }
gfCNCPoint1[5572] = {X 152.1286, Y 56.7358, Z -1.3333, A 0.000, B 0.000, C 0.000 }
gfCNCPoint1[5573] = {X 152.4570, Y 55.5101, Z -1.3333, A 0.000, B 0.000, C 0.000 }
gfCNCPoint1[5574] = {X 152.9933, Y 54.3600, Z -1.3333, A 0.000, B 0.000, C 0.000 }
gfCNCPoint1[5575] = {X 153.7212, Y 53.3205, Z -1.3333, A 0.000, B 0.000, C 0.000 }
gfCNCPoint1[5576] = {X 154.6185, Y 52.4232, Z -1.3333, A 0.000, B 0.000, C 0.000 }
gfCNCPoint1[5577] = {X 155.6580, Y 51.6953, Z -1.3333, A 0.000, B 0.000, C 0.000 }
gfCNCPoint1[5578] = {X 156.8081, Y 51.1590, Z -1.3333, A 0.000, B 0.000, C 0.000 }
gfCNCPoint1[5579] = {X 158.0338, Y 50.8306, Z -1.3333, A 0.000, B 0.000, C 0.000 }
gfCNCPoint1[5580] = {X 159.2980, Y 50.7200, Z -1.3333, A 0.000, B 0.000, C 0.000 }
gfCNCPoint1[5581] = {X 178.5335, Y 50.7200, Z -1.3333, A 0.000, B 0.000, C 0.000 }
gfCNCPoint1[5582] = {X 179.7860, Y 50.8286, Z -1.3333, A 0.000, B 0.000, C 0.000 }
gfCNCPoint1[5583] = {X 181.0012, Y 51.1510, Z -1.3333, A 0.000, B 0.000, C 0.000 }
gfCNCPoint1[5584] = {X 182.1427, Y 51.6777, Z -1.3333, A 0.000, B 0.000, C 0.000 }
gfCNCPoint1[5585] = {X 183.1767, Y 52.3929, Z -1.3333, A 0.000, B 0.000, C 0.000 }
gfCNCPoint1[5586] = {X 184.0859, Y 53.2916, Z -1.3333, A 0.000, B 0.000, C 0.000 }
gfCNCPoint1[5587] = {X 184.8239, Y 54.3355, Z -1.3333, A 0.000, B 0.000, C 0.000 }
gfCNCPoint1[5588] = {X 185.3680, Y 55.4923, Z -1.3333, A 0.000, B 0.000, C 0.000 }
gfCNCPoint1[5589] = {X 185.7013, Y 56.7265, Z -1.3333, A 0.000, B 0.000, C 0.000 }
gfCNCPoint1[5590] = {X 185.8135, Y 58.0000, Z -1.3333, A 0.000, B 0.000, C 0.000 }
gfCNCPoint1[5591] = {X 185.8133, Y 58.9942, Z -1.3333, A 0.000, B 0.000, C 0.000 }
gfCNCPoint1[5592] = {X 185.7647, Y 59.7756, Z -1.3333, A 0.000, B 0.000, C 0.000 }
gfCNCPoint1[5593] = {X 185.6325, Y 60.5472, Z -1.3333, A 0.000, B 0.000, C 0.000 }
gfCNCPoint1[5594] = {X 211.6596, Y 88.9542, Z -1.3333, A 0.000, B 0.000, C 0.000 }
gfCNCPoint1[5595] = {X 212.0306, Y 89.3378, Z -1.3333, A 0.000, B 0.000, C 0.000 }
gfCNCPoint1[5596] = {X 212.4216, Y 89.7009, Z -1.3333, A 0.000, B 0.000, C 0.000 }
gfCNCPoint1[5597] = {X 212.9250, Y 89.7845, Z -1.3333, A 0.000, B 0.000, C 0.000 }
gfCNCPoint1[5598] = {X 213.4317, Y 89.8454, Z -1.3333, A 0.000, B 0.000, C 0.000 }
gfCNCPoint1[5599] = {X 214.4177, Y 89.7737, Z -1.3333, A 0.000, B 0.000, C 0.000 }
gfCNCPoint1[5600] = {X 215.4047, Y 89.7184, Z -1.3333, A 0.000, B 0.000, C 0.000 }
gfCNCPoint1[5601] = {X 215.6222, Y 89.6959, Z -1.3333, A 0.000, B 0.000, C 0.000 }
gfCNCPoint1[5602] = {X 215.8222, Y 89.6074, Z -1.3333, A 0.000, B 0.000, C 0.000 }
gfCNCPoint1[5603] = {X 239.3478, Y 74.5355, Z -1.3333, A 0.000, B 0.000, C 0.000 }
gfCNCPoint1[5604] = {X 220.5435, Y 67.1556, Z -1.3333, A 0.000, B 0.000, C 0.000 }
gfCNCPoint1[5605] = {X 219.0954, Y 66.6695, Z -1.3333, A 0.000, B 0.000, C 0.000 }
gfCNCPoint1[5606] = {X 217.6011, Y 66.3528, Z -1.3333, A 0.000, B 0.000, C 0.000 }
gfCNCPoint1[5607] = {X 216.0803, Y 66.2098, Z -1.3333, A 0.000, B 0.000, C 0.000 }
gfCNCPoint1[5608] = {X 214.8534, Y 66.0626, Z -1.3333, A 0.000, B 0.000, C 0.000 }
gfCNCPoint1[5609] = {X 213.6691, Y 65.7100, Z -1.3333, A 0.000, B 0.000, C 0.000 }
gfCNCPoint1[5610] = {X 212.5615, Y 65.1623, Z -1.3333, A 0.000, B 0.000, C 0.000 }
gfCNCPoint1[5611] = {X 211.5624, Y 64.4351, Z -1.3333, A 0.000, B 0.000, C 0.000 }
gfCNCPoint1[5612] = {X 210.7008, Y 63.5494, Z -1.3333, A 0.000, B 0.000, C 0.000 }
gfCNCPoint1[5613] = {X 210.0013, Y 62.5308, Z -1.3333, A 0.000, B 0.000, C 0.000 }
gfCNCPoint1[5614] = {X 209.4842, Y 61.4085, Z -1.3333, A 0.000, B 0.000, C 0.000 }
gfCNCPoint1[5615] = {X 209.1644, Y 60.2149, Z -1.3333, A 0.000, B 0.000, C 0.000 }
gfCNCPoint1[5616] = {X 209.0510, Y 58.9845, Z -1.3333, A 0.000, B 0.000, C 0.000 }
gfCNCPoint1[5617] = {X 209.0508, Y 58.0000, Z -1.3333, A 0.000, B 0.000, C 0.000 }
gfCNCPoint1[5618] = {X 209.1477, Y 56.8162, Z -1.3333, A 0.000, B 0.000, C 0.000 }
gfCNCPoint1[5619] = {X 209.4358, Y 55.6638, Z -1.3333, A 0.000, B 0.000, C 0.000 }
gfCNCPoint1[5620] = {X 209.9075, Y 54.5737, Z -1.3333, A 0.000, B 0.000, C 0.000 }
gfCNCPoint1[5621] = {X 210.5502, Y 53.5748, Z -1.3333, A 0.000, B 0.000, C 0.000 }
gfCNCPoint1[5622] = {X 211.3467, Y 52.6937, Z -1.3333, A 0.000, B 0.000, C 0.000 }
gfCNCPoint1[5623] = {X 212.2759, Y 51.9538, Z -1.3333, A 0.000, B 0.000, C 0.000 }
gfCNCPoint1[5624] = {X 213.3131, Y 51.3749, Z -1.3333, A 0.000, B 0.000, C 0.000 }
gfCNCPoint1[5625] = {X 214.4306, Y 50.9724, Z -1.3333, A 0.000, B 0.000, C 0.000 }
gfCNCPoint1[5626] = {X 215.3724, Y 50.7834, Z -1.3333, A 0.000, B 0.000, C 0.000 }
gfCNCPoint1[5627] = {X 216.3308, Y 50.7200, Z -1.3333, A 0.000, B 0.000, C 0.000 }
gfCNCPoint1[5628] = {X 237.2617, Y 50.7200, Z -1.3333, A 0.000, B 0.000, C 0.000 }
gfCNCPoint1[5629] = {X 238.3057, Y 50.7953, Z -1.3333, A 0.000, B 0.000, C 0.000 }
gfCNCPoint1[5630] = {X 239.3282, Y 51.0195, Z -1.3333, A 0.000, B 0.000, C 0.000 }
gfCNCPoint1[5631] = {X 240.3080, Y 51.3880, Z -1.3333, A 0.000, B 0.000, C 0.000 }
gfCNCPoint1[5632] = {X 241.2247, Y 51.8932, Z -1.3333, A 0.000, B 0.000, C 0.000 }
gfCNCPoint1[5633] = {X 242.0742, Y 52.5376, Z -1.3333, A 0.000, B 0.000, C 0.000 }
gfCNCPoint1[5634] = {X 242.8205, Y 53.2992, Z -1.3333, A 0.000, B 0.000, C 0.000 }
gfCNCPoint1[5635] = {X 243.4475, Y 54.1615, Z -1.3333, A 0.000, B 0.000, C 0.000 }
gfCNCPoint1[5636] = {X 243.9419, Y 55.1063, Z -1.3333, A 0.000, B 0.000, C 0.000 }
gfCNCPoint1[5637] = {X 244.2929, Y 56.1131, Z -1.3333, A 0.000, B 0.000, C 0.000 }
gfCNCPoint1[5638] = {X 249.2018, Y 58.0270, Z -1.3333, A 0.000, B 0.000, C 0.000 }
gfCNCPoint1[5639] = {X 272.6737, Y 67.3435, Z -1.3333, A 0.000, B 0.000, C 0.000 }
gfCNCPoint1[5640] = {X 272.6735, Y 65.2847, Z -1.3333, A 0.000, B 0.000, C 0.000 }
gfCNCPoint1[5641] = {X 271.6657, Y 64.6034, Z -1.3333, A 0.000, B 0.000, C 0.000 }
gfCNCPoint1[5642] = {X 270.7855, Y 63.7638, Z -1.3333, A 0.000, B 0.000, C 0.000 }
gfCNCPoint1[5643] = {X 270.0573, Y 62.7893, Z -1.3333, A 0.000, B 0.000, C 0.000 }
gfCNCPoint1[5644] = {X 269.5016, Y 61.7072, Z -1.3333, A 0.000, B 0.000, C 0.000 }
gfCNCPoint1[5645] = {X 269.2027, Y 60.8256, Z -1.3333, A 0.000, B 0.000, C 0.000 }
gfCNCPoint1[5646] = {X 269.0188, Y 59.9130, Z -1.3333, A 0.000, B 0.000, C 0.000 }
gfCNCPoint1[5647] = {X 268.9529, Y 58.9845, Z -1.3333, A 0.000, B 0.000, C 0.000 }
gfCNCPoint1[5648] = {X 268.9527, Y 58.0000, Z -1.3333, A 0.000, B 0.000, C 0.000 }
gfCNCPoint1[5649] = {X 269.0633, Y 56.7358, Z -1.3333, A 0.000, B 0.000, C 0.000 }
gfCNCPoint1[5650] = {X 269.3917, Y 55.5101, Z -1.3333, A 0.000, B 0.000, C 0.000 }
gfCNCPoint1[5651] = {X 269.9280, Y 54.3600, Z -1.3333, A 0.000, B 0.000, C 0.000 }
gfCNCPoint1[5652] = {X 270.6559, Y 53.3205, Z -1.3333, A 0.000, B 0.000, C 0.000 }
gfCNCPoint1[5653] = {X 271.5532, Y 52.4232, Z -1.3333, A 0.000, B 0.000, C 0.000 }
gfCNCPoint1[5654] = {X 272.5927, Y 51.6953, Z -1.3333, A 0.000, B 0.000, C 0.000 }
gfCNCPoint1[5655] = {X 273.7428, Y 51.1590, Z -1.3333, A 0.000, B 0.000, C 0.000 }
gfCNCPoint1[5656] = {X 274.9685, Y 50.8306, Z -1.3333, A 0.000, B 0.000, C 0.000 }
gfCNCPoint1[5657] = {X 276.2327, Y 50.7200, Z -1.3333, A 0.000, B 0.000, C 0.000 }
gfCNCPoint1[5658] = {X 292.7731, Y 50.7200, Z -1.3333, A 0.000, B 0.000, C 0.000 }
gfCNCPoint1[5659] = {X 293.4209, Y 50.7489, Z -1.3333, A 0.000, B 0.000, C 0.000 }
gfCNCPoint1[5660] = {X 294.0636, Y 50.8353, Z -1.3333, A 0.000, B 0.000, C 0.000 }
gfCNCPoint1[5661] = {X 294.7296, Y 50.9878, Z -1.3333, A 0.000, B 0.000, C 0.000 }
gfCNCPoint1[5662] = {X 295.3785, Y 51.2022, Z -1.3333, A 0.000, B 0.000, C 0.000 }
gfCNCPoint1[5663] = {X 298.3088, Y 43.5563, Z -1.3333, A 0.000, B 0.000, C 0.000 }
gfCNCPoint1[5664] = {X 298.4822, Y 42.5321, Z -1.3333, A 0.000, B 0.000, C 0.000 }
gfCNCPoint1[5665] = {X 298.7930, Y 41.5409, Z -1.3333, A 0.000, B 0.000, C 0.000 }
gfCNCPoint1[5666] = {X 299.2353, Y 40.6010, Z -1.3333, A 0.000, B 0.000, C 0.000 }
gfCNCPoint1[5667] = {X 299.8011, Y 39.7298, Z -1.3333, A 0.000, B 0.000, C 0.000 }
gfCNCPoint1[5668] = {X 299.8011, Y 36.9943, Z -1.3333, A 0.000, B 0.000, C 0.000 }
gfCNCPoint1[5669] = {X 296.8131, Y 36.9943, Z -1.3333, A 0.000, B 0.000, C 0.000 }
gfCNCPoint1[5670] = {X 296.8126, Y 39.7493, Z -1.3333, A 0.000, B 0.000, C 0.000 }
gfCNCPoint1[5671] = {X 297.3843, Y 40.6124, Z -1.3333, A 0.000, B 0.000, C 0.000 }
gfCNCPoint1[5672] = {X 297.8296, Y 41.5471, Z -1.3333, A 0.000, B 0.000, C 0.000 }
gfCNCPoint1[5673] = {X 298.1399, Y 42.5349, Z -1.3333, A 0.000, B 0.000, C 0.000 }
gfCNCPoint1[5674] = {X 298.3088, Y 43.5563, Z -1.3333, A 0.000, B 0.000, C 0.000 }
gfCNCPoint1[5675] = {X 296.2374, Y 48.9611, Z -1.3333, A 0.000, B 0.000, C 0.000 }
gfCNCPoint1[5676] = {X 296.6129, Y 49.1142, Z -1.3333, A 0.000, B 0.000, C 0.000 }
gfCNCPoint1[5677] = {X 296.9817, Y 49.2828, Z -1.3333, A 0.000, B 0.000, C 0.000 }
gfCNCPoint1[5678] = {X 297.2571, Y 49.4212, Z -1.3333, A 0.000, B 0.000, C 0.000 }
gfCNCPoint1[5679] = {X 297.5280, Y 49.5683, Z -1.3333, A 0.000, B 0.000, C 0.000 }
gfCNCPoint1[5680] = {X 298.7174, Y 50.3602, Z -1.3333, A 0.000, B 0.000, C 0.000 }
gfCNCPoint1[5681] = {X 299.7774, Y 51.3185, Z -1.3333, A 0.000, B 0.000, C 0.000 }
gfCNCPoint1[5682] = {X 300.6847, Y 52.4224, Z -1.3333, A 0.000, B 0.000, C 0.000 }
gfCNCPoint1[5683] = {X 301.5914, Y 51.3191, Z -1.3333, A 0.000, B 0.000, C 0.000 }
gfCNCPoint1[5684] = {X 302.6506, Y 50.3611, Z -1.3333, A 0.000, B 0.000, C 0.000 }
gfCNCPoint1[5685] = {X 303.8393, Y 49.5695, Z -1.3333, A 0.000, B 0.000, C 0.000 }
gfCNCPoint1[5686] = {X 302.8989, Y 49.0956, Z -1.3333, A 0.000, B 0.000, C 0.000 }
gfCNCPoint1[5687] = {X 302.0820, Y 48.4310, Z -1.3333, A 0.000, B 0.000, C 0.000 }
gfCNCPoint1[5688] = {X 301.4268, Y 47.6067, Z -1.3333, A 0.000, B 0.000, C 0.000 }
gfCNCPoint1[5689] = {X 300.9636, Y 46.6610, Z -1.3333, A 0.000, B 0.000, C 0.000 }
gfCNCPoint1[5690] = {X 300.7923, Y 46.0759, Z -1.3333, A 0.000, B 0.000, C 0.000 }
gfCNCPoint1[5691] = {X 300.6953, Y 45.4741, Z -1.3333, A 0.000, B 0.000, C 0.000 }
gfCNCPoint1[5692] = {X 300.6790, Y 45.2570, Z -1.3333, A 0.000, B 0.000, C 0.000 }
gfCNCPoint1[5693] = {X 300.6724, Y 45.0393, Z -1.3333, A 0.000, B 0.000, C 0.000 }
gfCNCPoint1[5694] = {X 300.6725, Y 44.1872, Z -1.3333, A 0.000, B 0.000, C 0.000 }
gfCNCPoint1[5695] = {X 300.6811, Y 43.9910, Z -1.3333, A 0.000, B 0.000, C 0.000 }
gfCNCPoint1[5696] = {X 300.6969, Y 43.7952, Z -1.3333, A 0.000, B 0.000, C 0.000 }
gfCNCPoint1[5697] = {X 300.8619, Y 42.9149, Z -1.3333, A 0.000, B 0.000, C 0.000 }
gfCNCPoint1[5698] = {X 301.1743, Y 42.0756, Z -1.3333, A 0.000, B 0.000, C 0.000 }
gfCNCPoint1[5699] = {X 301.6251, Y 41.3018, Z -1.3333, A 0.000, B 0.000, C 0.000 }
gfCNCPoint1[5700] = {X 302.2011, Y 40.6161, Z -1.3333, A 0.000, B 0.000, C 0.000 }
gfCNCPoint1[5701] = {X 302.2011, Y 34.5943, Z -1.3333, A 0.000, B 0.000, C 0.000 }
gfCNCPoint1[5702] = {X 294.4134, Y 34.5943, Z -1.3333, A 0.000, B 0.000, C 0.000 }
gfCNCPoint1[5703] = {X 294.4125, Y 40.6561, Z -1.3333, A 0.000, B 0.000, C 0.000 }
gfCNCPoint1[5704] = {X 294.9932, Y 41.3236, Z -1.3333, A 0.000, B 0.000, C 0.000 }
gfCNCPoint1[5705] = {X 295.4467, Y 42.0832, Z -1.3333, A 0.000, B 0.000, C 0.000 }
gfCNCPoint1[5706] = {X 295.7587, Y 42.9111, Z -1.3333, A 0.000, B 0.000, C 0.000 }
gfCNCPoint1[5707] = {X 295.9194, Y 43.7811, Z -1.3333, A 0.000, B 0.000, C 0.000 }
gfCNCPoint1[5708] = {X 295.9349, Y 43.9948, Z -1.3333, A 0.000, B 0.000, C 0.000 }
gfCNCPoint1[5709] = {X 295.9411, Y 44.2089, Z -1.3333, A 0.000, B 0.000, C 0.000 }
gfCNCPoint1[5710] = {X 295.9411, Y 45.0000, Z -1.3333, A 0.000, B 0.000, C 0.000 }
gfCNCPoint1[5711] = {X 295.9354, Y 45.2373, Z -1.3333, A 0.000, B 0.000, C 0.000 }
gfCNCPoint1[5712] = {X 295.9180, Y 45.4741, Z -1.3333, A 0.000, B 0.000, C 0.000 }
gfCNCPoint1[5713] = {X 298.3067, Y 45.7073, Z -1.3333, A 0.000, B 0.000, C 0.000 }
gfCNCPoint1[5714] = {X 298.2010, Y 46.4214, Z -1.3333, A 0.000, B 0.000, C 0.000 }
gfCNCPoint1[5715] = {X 298.0252, Y 47.1215, Z -1.3333, A 0.000, B 0.000, C 0.000 }
gfCNCPoint1[5716] = {X 298.3689, Y 47.2942, Z -1.3333, A 0.000, B 0.000, C 0.000 }
gfCNCPoint1[5717] = {X 298.7069, Y 47.4778, Z -1.3333, A 0.000, B 0.000, C 0.000 }
gfCNCPoint1[5718] = {X 298.4514, Y 46.6051, Z -1.3333, A 0.000, B 0.000, C 0.000 }
gfCNCPoint1[5719] = {X 298.3067, Y 45.7073, Z -1.3333, A 0.000, B 0.000, C 0.000 }
gfCNCPoint1[5720] = {X 295.9180, Y 45.4741, Z -1.3333, A 0.000, B 0.000, C 0.000 }
gfCNCPoint1[5721] = {X 295.8472, Y 45.9528, Z -1.3333, A 0.000, B 0.000, C 0.000 }
gfCNCPoint1[5722] = {X 295.7293, Y 46.4221, Z -1.3333, A 0.000, B 0.000, C 0.000 }
gfCNCPoint1[5723] = {X 295.4314, Y 47.1714, Z -1.3333, A 0.000, B 0.000, C 0.000 }
gfCNCPoint1[5724] = {X 295.0142, Y 47.8614, Z -1.3333, A 0.000, B 0.000, C 0.000 }
gfCNCPoint1[5725] = {X 294.4890, Y 48.4733, Z -1.3333, A 0.000, B 0.000, C 0.000 }
gfCNCPoint1[5726] = {X 295.3747, Y 48.6762, Z -1.3333, A 0.000, B 0.000, C 0.000 }
gfCNCPoint1[5727] = {X 296.2374, Y 48.9611, Z -1.3333, A 0.000, B 0.000, C 0.000 }
gfCNCPoint1[5728] = {X 295.3785, Y 51.2022, Z -1.3333, A 0.000, B 0.000, C 0.000 }
gfCNCPoint1[5729] = {X 296.3504, Y 51.6595, Z -1.3333, A 0.000, B 0.000, C 0.000 }
gfCNCPoint1[5730] = {X 297.2444, Y 52.2549, Z -1.3333, A 0.000, B 0.000, C 0.000 }
gfCNCPoint1[5731] = {X 298.0411, Y 52.9754, Z -1.3333, A 0.000, B 0.000, C 0.000 }
gfCNCPoint1[5732] = {X 298.7231, Y 53.8053, Z -1.3333, A 0.000, B 0.000, C 0.000 }
gfCNCPoint1[5733] = {X 299.2946, Y 54.7645, Z -1.3333, A 0.000, B 0.000, C 0.000 }
gfCNCPoint1[5734] = {X 299.7126, Y 55.7997, Z -1.3333, A 0.000, B 0.000, C 0.000 }
gfCNCPoint1[5735] = {X 299.9675, Y 56.8868, Z -1.3333, A 0.000, B 0.000, C 0.000 }
gfCNCPoint1[5736] = {X 300.0531, Y 58.0000, Z -1.3333, A 0.000, B 0.000, C 0.000 }
gfCNCPoint1[5737] = {X 300.0531, Y 58.9458, Z -1.3333, A 0.000, B 0.000, C 0.000 }
gfCNCPoint1[5738] = {X 299.9643, Y 60.0549, Z -1.3333, A 0.000, B 0.000, C 0.000 }
gfCNCPoint1[5739] = {X 299.7079, Y 61.1376, Z -1.3333, A 0.000, B 0.000, C 0.000 }
gfCNCPoint1[5740] = {X 299.2899, Y 62.1687, Z -1.3333, A 0.000, B 0.000, C 0.000 }
gfCNCPoint1[5741] = {X 298.7200, Y 63.1243, Z -1.3333, A 0.000, B 0.000, C 0.000 }
gfCNCPoint1[5742] = {X 300.6815, Y 64.5072, Z -1.3333, A 0.000, B 0.000, C 0.000 }
gfCNCPoint1[5743] = {X 299.7816, Y 65.6036, Z -1.3333, A 0.000, B 0.000, C 0.000 }
gfCNCPoint1[5744] = {X 298.7314, Y 66.5570, Z -1.3333, A 0.000, B 0.000, C 0.000 }
gfCNCPoint1[5745] = {X 298.7314, Y 89.4425, Z -1.3333, A 0.000, B 0.000, C 0.000 }
gfCNCPoint1[5746] = {X 299.8282, Y 90.4467, Z -1.3333, A 0.000, B 0.000, C 0.000 }
gfCNCPoint1[5747] = {X 300.7589, Y 91.6066, Z -1.3333, A 0.000, B 0.000, C 0.000 }
gfCNCPoint1[5748] = {X 301.5016, Y 92.8949, Z -1.3333, A 0.000, B 0.000, C 0.000 }
gfCNCPoint1[5749] = {X 304.0687, Y 92.8949, Z -1.3333, A 0.000, B 0.000, C 0.000 }
gfCNCPoint1[5750] = {X 303.7112, Y 91.9005, Z -1.3333, A 0.000, B 0.000, C 0.000 }
gfCNCPoint1[5751] = {X 303.4152, Y 90.8861, Z -1.3333, A 0.000, B 0.000, C 0.000 }
gfCNCPoint1[5752] = {X 302.9758, Y 88.8143, Z -1.3333, A 0.000, B 0.000, C 0.000 }
gfCNCPoint1[5753] = {X 302.7157, Y 86.7125, Z -1.3333, A 0.000, B 0.000, C 0.000 }
gfCNCPoint1[5754] = {X 302.6367, Y 84.5962, Z -1.3333, A 0.000, B 0.000, C 0.000 }
gfCNCPoint1[5755] = {X 302.6380, Y 83.2276, Z -1.3333, A 0.000, B 0.000, C 0.000 }
gfCNCPoint1[5756] = {X 302.6380, Y 66.5631, Z -1.3333, A 0.000, B 0.000, C 0.000 }
gfCNCPoint1[5757] = {X 301.5840, Y 65.6072, Z -1.3333, A 0.000, B 0.000, C 0.000 }
gfCNCPoint1[5758] = {X 300.6815, Y 64.5072, Z -1.3333, A 0.000, B 0.000, C 0.000 }
gfCNCPoint1[5759] = {X 298.7200, Y 63.1243, Z -1.3333, A 0.000, B 0.000, C 0.000 }
gfCNCPoint1[5760] = {X 298.0337, Y 63.9590, Z -1.3333, A 0.000, B 0.000, C 0.000 }
gfCNCPoint1[5761] = {X 297.2316, Y 64.6831, Z -1.3333, A 0.000, B 0.000, C 0.000 }
gfCNCPoint1[5762] = {X 296.3314, Y 65.2808, Z -1.3333, A 0.000, B 0.000, C 0.000 }
gfCNCPoint1[5763] = {X 296.3314, Y 90.7171, Z -1.3333, A 0.000, B 0.000, C 0.000 }
gfCNCPoint1[5764] = {X 297.3117, Y 91.3796, Z -1.3333, A 0.000, B 0.000, C 0.000 }
gfCNCPoint1[5765] = {X 298.1723, Y 92.1915, Z -1.3333, A 0.000, B 0.000, C 0.000 }
gfCNCPoint1[5766] = {X 298.8907, Y 93.1315, Z -1.3333, A 0.000, B 0.000, C 0.000 }
gfCNCPoint1[5767] = {X 299.4481, Y 94.1751, Z -1.3333, A 0.000, B 0.000, C 0.000 }
gfCNCPoint1[5768] = {X 299.8300, Y 95.2949, Z -1.3333, A 0.000, B 0.000, C 0.000 }
gfCNCPoint1[5769] = {X 308.1008, Y 95.2949, Z -1.3333, A 0.000, B 0.000, C 0.000 }
gfCNCPoint1[5770] = {X 307.0976, Y 93.7114, Z -1.3333, A 0.000, B 0.000, C 0.000 }
gfCNCPoint1[5771] = {X 306.3013, Y 92.0143, Z -1.3333, A 0.000, B 0.000, C 0.000 }
gfCNCPoint1[5772] = {X 305.9935, Y 91.1580, Z -1.3333, A 0.000, B 0.000, C 0.000 }
gfCNCPoint1[5773] = {X 305.7385, Y 90.2844, Z -1.3333, A 0.000, B 0.000, C 0.000 }
gfCNCPoint1[5774] = {X 305.3421, Y 88.4135, Z -1.3333, A 0.000, B 0.000, C 0.000 }
gfCNCPoint1[5775] = {X 305.1076, Y 86.5154, Z -1.3333, A 0.000, B 0.000, C 0.000 }
gfCNCPoint1[5776] = {X 305.0367, Y 84.6043, Z -1.3333, A 0.000, B 0.000, C 0.000 }
gfCNCPoint1[5777] = {X 305.0380, Y 83.2289, Z -1.3333, A 0.000, B 0.000, C 0.000 }
gfCNCPoint1[5778] = {X 305.0380, Y 65.2852, Z -1.3333, A 0.000, B 0.000, C 0.000 }
gfCNCPoint1[5779] = {X 304.1353, Y 64.6872, Z -1.3333, A 0.000, B 0.000, C 0.000 }
gfCNCPoint1[5780] = {X 303.3313, Y 63.9619, Z -1.3333, A 0.000, B 0.000, C 0.000 }
gfCNCPoint1[5781] = {X 302.6438, Y 63.1254, Z -1.3333, A 0.000, B 0.000, C 0.000 }
gfCNCPoint1[5782] = {X 302.0790, Y 62.1781, Z -1.3333, A 0.000, B 0.000, C 0.000 }
gfCNCPoint1[5783] = {X 301.6637, Y 61.1564, Z -1.3333, A 0.000, B 0.000, C 0.000 }
gfCNCPoint1[5784] = {X 301.4076, Y 60.0836, Z -1.3333, A 0.000, B 0.000, C 0.000 }
gfCNCPoint1[5785] = {X 301.3164, Y 58.9845, Z -1.3333, A 0.000, B 0.000, C 0.000 }
gfCNCPoint1[5786] = {X 301.3162, Y 58.0000, Z -1.3333, A 0.000, B 0.000, C 0.000 }
gfCNCPoint1[5787] = {X 301.4018, Y 56.8868, Z -1.3333, A 0.000, B 0.000, C 0.000 }
gfCNCPoint1[5788] = {X 301.6567, Y 55.7997, Z -1.3333, A 0.000, B 0.000, C 0.000 }
gfCNCPoint1[5789] = {X 302.0747, Y 54.7645, Z -1.3333, A 0.000, B 0.000, C 0.000 }
gfCNCPoint1[5790] = {X 302.6462, Y 53.8053, Z -1.3333, A 0.000, B 0.000, C 0.000 }
gfCNCPoint1[5791] = {X 303.3281, Y 52.9755, Z -1.3333, A 0.000, B 0.000, C 0.000 }
gfCNCPoint1[5792] = {X 304.1247, Y 52.2551, Z -1.3333, A 0.000, B 0.000, C 0.000 }
gfCNCPoint1[5793] = {X 305.0187, Y 51.6597, Z -1.3333, A 0.000, B 0.000, C 0.000 }
gfCNCPoint1[5794] = {X 306.1514, Y 51.1428, Z -1.3333, A 0.000, B 0.000, C 0.000 }
gfCNCPoint1[5795] = {X 307.3557, Y 50.8265, Z -1.3333, A 0.000, B 0.000, C 0.000 }
gfCNCPoint1[5796] = {X 308.5962, Y 50.7200, Z -1.3333, A 0.000, B 0.000, C 0.000 }
gfCNCPoint1[5797] = {X 324.3107, Y 50.7200, Z -1.3333, A 0.000, B 0.000, C 0.000 }
gfCNCPoint1[5798] = {X 325.2469, Y 50.7804, Z -1.3333, A 0.000, B 0.000, C 0.000 }
gfCNCPoint1[5799] = {X 326.1675, Y 50.9608, Z -1.3333, A 0.000, B 0.000, C 0.000 }
gfCNCPoint1[5800] = {X 326.5260, Y 51.0653, Z -1.3333, A 0.000, B 0.000, C 0.000 }
gfCNCPoint1[5801] = {X 326.8787, Y 51.1880, Z -1.3333, A 0.000, B 0.000, C 0.000 }
gfCNCPoint1[5802] = {X 327.4582, Y 51.4356, Z -1.3333, A 0.000, B 0.000, C 0.000 }
gfCNCPoint1[5803] = {X 328.0140, Y 51.7323, Z -1.3333, A 0.000, B 0.000, C 0.000 }
gfCNCPoint1[5804] = {X 328.5423, Y 52.0762, Z -1.3333, A 0.000, B 0.000, C 0.000 }
gfCNCPoint1[5805] = {X 329.0389, Y 52.4644, Z -1.3333, A 0.000, B 0.000, C 0.000 }
gfCNCPoint1[5806] = {X 329.9201, Y 53.3597, Z -1.3333, A 0.000, B 0.000, C 0.000 }
gfCNCPoint1[5807] = {X 330.6344, Y 54.3932, Z -1.3333, A 0.000, B 0.000, C 0.000 }
gfCNCPoint1[5808] = {X 331.1603, Y 55.5341, Z -1.3333, A 0.000, B 0.000, C 0.000 }
gfCNCPoint1[5809] = {X 331.4823, Y 56.7484, Z -1.3333, A 0.000, B 0.000, C 0.000 }
gfCNCPoint1[5810] = {X 331.5907, Y 58.0000, Z -1.3333, A 0.000, B 0.000, C 0.000 }
gfCNCPoint1[5811] = {X 331.5907, Y 58.9403, Z -1.3333, A 0.000, B 0.000, C 0.000 }
gfCNCPoint1[5812] = {X 331.4729, Y 60.2171, Z -1.3333, A 0.000, B 0.000, C 0.000 }
gfCNCPoint1[5813] = {X 331.1341, Y 61.4537, Z -1.3333, A 0.000, B 0.000, C 0.000 }
gfCNCPoint1[5814] = {X 330.5847, Y 62.6122, Z -1.3333, A 0.000, B 0.000, C 0.000 }
gfCNCPoint1[5815] = {X 329.8416, Y 63.6571, Z -1.3333, A 0.000, B 0.000, C 0.000 }
gfCNCPoint1[5816] = {X 328.9276, Y 64.5563, Z -1.3333, A 0.000, B 0.000, C 0.000 }
gfCNCPoint1[5817] = {X 327.8707, Y 65.2822, Z -1.3333, A 0.000, B 0.000, C 0.000 }
gfCNCPoint1[5818] = {X 327.8719, Y 83.2150, Z -1.3333, A 0.000, B 0.000, C 0.000 }
gfCNCPoint1[5819] = {X 327.8854, Y 84.5926, Z -1.3333, A 0.000, B 0.000, C 0.000 }
gfCNCPoint1[5820] = {X 327.8946, Y 84.9548, Z -1.3333, A 0.000, B 0.000, C 0.000 }
gfCNCPoint1[5821] = {X 327.9215, Y 85.3161, Z -1.3333, A 0.000, B 0.000, C 0.000 }
gfCNCPoint1[5822] = {X 328.8632, Y 85.6740, Z -1.3333, A 0.000, B 0.000, C 0.000 }
gfCNCPoint1[5823] = {X 329.8334, Y 85.9457, Z -1.3333, A 0.000, B 0.000, C 0.000 }
gfCNCPoint1[5824] = {X 332.7087, Y 86.5217, Z -1.3333, A 0.000, B 0.000, C 0.000 }
gfCNCPoint1[5825] = {X 335.6182, Y 86.8881, Z -1.3333, A 0.000, B 0.000, C 0.000 }
gfCNCPoint1[5826] = {X 340.6718, Y 87.2624, Z -1.3333, A 0.000, B 0.000, C 0.000 }
gfCNCPoint1[5827] = {X 345.7373, Y 87.4033, Z -1.3333, A 0.000, B 0.000, C 0.000 }
gfCNCPoint1[5828] = {X 350.4845, Y 87.4099, Z -1.3333, A 0.000, B 0.000, C 0.000 }
gfCNCPoint1[5829] = {X 355.2288, Y 87.2451, Z -1.3333, A 0.000, B 0.000, C 0.000 }
gfCNCPoint1[5830] = {X 359.9641, Y 86.9089, Z -1.3333, A 0.000, B 0.000, C 0.000 }
gfCNCPoint1[5831] = {X 362.3288, Y 86.6411, Z -1.3333, A 0.000, B 0.000, C 0.000 }
gfCNCPoint1[5832] = {X 364.6716, Y 86.2236, Z -1.3333, A 0.000, B 0.000, C 0.000 }
gfCNCPoint1[5833] = {X 366.9833, Y 85.6582, Z -1.3333, A 0.000, B 0.000, C 0.000 }
gfCNCPoint1[5834] = {X 367.4436, Y 85.5117, Z -1.3333, A 0.000, B 0.000, C 0.000 }
gfCNCPoint1[5835] = {X 367.8901, Y 85.3273, Z -1.3333, A 0.000, B 0.000, C 0.000 }
gfCNCPoint1[5836] = {X 367.9436, Y 84.5784, Z -1.3333, A 0.000, B 0.000, C 0.000 }
gfCNCPoint1[5837] = {X 367.9614, Y 83.8279, Z -1.3333, A 0.000, B 0.000, C 0.000 }
gfCNCPoint1[5838] = {X 367.9598, Y 65.2846, Z -1.3333, A 0.000, B 0.000, C 0.000 }
gfCNCPoint1[5839] = {X 366.9057, Y 64.5655, Z -1.3333, A 0.000, B 0.000, C 0.000 }
gfCNCPoint1[5840] = {X 365.9933, Y 63.6735, Z -1.3333, A 0.000, B 0.000, C 0.000 }
gfCNCPoint1[5841] = {X 365.2507, Y 62.6358, Z -1.3333, A 0.000, B 0.000, C 0.000 }
gfCNCPoint1[5842] = {X 364.7006, Y 61.4845, Z -1.3333, A 0.000, B 0.000, C 0.000 }
gfCNCPoint1[5843] = {X 364.3601, Y 60.2548, Z -1.3333, A 0.000, B 0.000, C 0.000 }
gfCNCPoint1[5844] = {X 364.2395, Y 58.9845, Z -1.3333, A 0.000, B 0.000, C 0.000 }
gfCNCPoint1[5845] = {X 364.2393, Y 58.0000, Z -1.3333, A 0.000, B 0.000, C 0.000 }
gfCNCPoint1[5846] = {X 364.3499, Y 56.7358, Z -1.3333, A 0.000, B 0.000, C 0.000 }
gfCNCPoint1[5847] = {X 364.6783, Y 55.5101, Z -1.3333, A 0.000, B 0.000, C 0.000 }
gfCNCPoint1[5848] = {X 365.2146, Y 54.3600, Z -1.3333, A 0.000, B 0.000, C 0.000 }
gfCNCPoint1[5849] = {X 365.9425, Y 53.3205, Z -1.3333, A 0.000, B 0.000, C 0.000 }
gfCNCPoint1[5850] = {X 366.8398, Y 52.4232, Z -1.3333, A 0.000, B 0.000, C 0.000 }
gfCNCPoint1[5851] = {X 367.8793, Y 51.6953, Z -1.3333, A 0.000, B 0.000, C 0.000 }
gfCNCPoint1[5852] = {X 369.0294, Y 51.1590, Z -1.3333, A 0.000, B 0.000, C 0.000 }
gfCNCPoint1[5853] = {X 370.2551, Y 50.8306, Z -1.3333, A 0.000, B 0.000, C 0.000 }
gfCNCPoint1[5854] = {X 371.5193, Y 50.7200, Z -1.3333, A 0.000, B 0.000, C 0.000 }
gfCNCPoint1[5855] = {X 388.0597, Y 50.7200, Z -1.3333, A 0.000, B 0.000, C 0.000 }
gfCNCPoint1[5856] = {X 389.2271, Y 50.8142, Z -1.3333, A 0.000, B 0.000, C 0.000 }
gfCNCPoint1[5857] = {X 390.3643, Y 51.0944, Z -1.3333, A 0.000, B 0.000, C 0.000 }
gfCNCPoint1[5858] = {X 391.4418, Y 51.5533, Z -1.3333, A 0.000, B 0.000, C 0.000 }
gfCNCPoint1[5859] = {X 392.4319, Y 52.1791, Z -1.3333, A 0.000, B 0.000, C 0.000 }
gfCNCPoint1[5860] = {X 393.3087, Y 52.9556, Z -1.3333, A 0.000, B 0.000, C 0.000 }
gfCNCPoint1[5861] = {X 394.1855, Y 52.1791, Z -1.3333, A 0.000, B 0.000, C 0.000 }
gfCNCPoint1[5862] = {X 395.1756, Y 51.5533, Z -1.3333, A 0.000, B 0.000, C 0.000 }
gfCNCPoint1[5863] = {X 396.2531, Y 51.0944, Z -1.3333, A 0.000, B 0.000, C 0.000 }
gfCNCPoint1[5864] = {X 397.3903, Y 50.8142, Z -1.3333, A 0.000, B 0.000, C 0.000 }
gfCNCPoint1[5865] = {X 398.5577, Y 50.7200, Z -1.3333, A 0.000, B 0.000, C 0.000 }
gfCNCPoint1[5866] = {X 419.4886, Y 50.7200, Z -1.3333, A 0.000, B 0.000, C 0.000 }
gfCNCPoint1[5867] = {X 420.6741, Y 50.8172, Z -1.3333, A 0.000, B 0.000, C 0.000 }
gfCNCPoint1[5868] = {X 421.8279, Y 51.1061, Z -1.3333, A 0.000, B 0.000, C 0.000 }
gfCNCPoint1[5869] = {X 422.9193, Y 51.5791, Z -1.3333, A 0.000, B 0.000, C 0.000 }
gfCNCPoint1[5870] = {X 423.9191, Y 52.2234, Z -1.3333, A 0.000, B 0.000, C 0.000 }
gfCNCPoint1[5871] = {X 424.8006, Y 53.0220, Z -1.3333, A 0.000, B 0.000, C 0.000 }
gfCNCPoint1[5872] = {X 425.5404, Y 53.9535, Z -1.3333, A 0.000, B 0.000, C 0.000 }
gfCNCPoint1[5873] = {X 426.1185, Y 54.9929, Z -1.3333, A 0.000, B 0.000, C 0.000 }
gfCNCPoint1[5874] = {X 426.5197, Y 56.1127, Z -1.3333, A 0.000, B 0.000, C 0.000 }
gfCNCPoint1[5875] = {X 430.7006, Y 57.7423, Z -1.3333, A 0.000, B 0.000, C 0.000 }
gfCNCPoint1[5876] = {X 454.9007, Y 67.3435, Z -1.3333, A 0.000, B 0.000, C 0.000 }
gfCNCPoint1[5877] = {X 454.9004, Y 65.2847, Z -1.3333, A 0.000, B 0.000, C 0.000 }
gfCNCPoint1[5878] = {X 453.8928, Y 64.6035, Z -1.3333, A 0.000, B 0.000, C 0.000 }
gfCNCPoint1[5879] = {X 453.0127, Y 63.7642, Z -1.3333, A 0.000, B 0.000, C 0.000 }
gfCNCPoint1[5880] = {X 452.2846, Y 62.7900, Z -1.3333, A 0.000, B 0.000, C 0.000 }
gfCNCPoint1[5881] = {X 451.7289, Y 61.7082, Z -1.3333, A 0.000, B 0.000, C 0.000 }
gfCNCPoint1[5882] = {X 451.4298, Y 60.8263, Z -1.3333, A 0.000, B 0.000, C 0.000 }
gfCNCPoint1[5883] = {X 451.2458, Y 59.9134, Z -1.3333, A 0.000, B 0.000, C 0.000 }
gfCNCPoint1[5884] = {X 451.1798, Y 58.9845, Z -1.3333, A 0.000, B 0.000, C 0.000 }
gfCNCPoint1[5885] = {X 451.1796, Y 58.0000, Z -1.3333, A 0.000, B 0.000, C 0.000 }
gfCNCPoint1[5886] = {X 451.2795, Y 56.7981, Z -1.3333, A 0.000, B 0.000, C 0.000 }
gfCNCPoint1[5887] = {X 451.5765, Y 55.6291, Z -1.3333, A 0.000, B 0.000, C 0.000 }
gfCNCPoint1[5888] = {X 452.0624, Y 54.5253, Z -1.3333, A 0.000, B 0.000, C 0.000 }
gfCNCPoint1[5889] = {X 452.7238, Y 53.5168, Z -1.3333, A 0.000, B 0.000, C 0.000 }
gfCNCPoint1[5890] = {X 453.5427, Y 52.6313, Z -1.3333, A 0.000, B 0.000, C 0.000 }
gfCNCPoint1[5891] = {X 454.4966, Y 51.8932, Z -1.3333, A 0.000, B 0.000, C 0.000 }
gfCNCPoint1[5892] = {X 455.4133, Y 51.3880, Z -1.3333, A 0.000, B 0.000, C 0.000 }
gfCNCPoint1[5893] = {X 456.3931, Y 51.0195, Z -1.3333, A 0.000, B 0.000, C 0.000 }
gfCNCPoint1[5894] = {X 457.4155, Y 50.7953, Z -1.3333, A 0.000, B 0.000, C 0.000 }
gfCNCPoint1[5895] = {X 458.4596, Y 50.7200, Z -1.3333, A 0.000, B 0.000, C 0.000 }
gfCNCPoint1[5896] = {X 475.0000, Y 50.7200, Z -1.3333, A 0.000, B 0.000, C 0.000 }
gfCNCPoint1[5897] = {X 476.0441, Y 50.7953, Z -1.3333, A 0.000, B 0.000, C 0.000 }
gfCNCPoint1[5898] = {X 477.0665, Y 51.0195, Z -1.3333, A 0.000, B 0.000, C 0.000 }
gfCNCPoint1[5899] = {X 478.0463, Y 51.3880, Z -1.3333, A 0.000, B 0.000, C 0.000 }
gfCNCPoint1[5900] = {X 478.9630, Y 51.8932, Z -1.3333, A 0.000, B 0.000, C 0.000 }
gfCNCPoint1[5901] = {X 479.9169, Y 52.6313, Z -1.3333, A 0.000, B 0.000, C 0.000 }
gfCNCPoint1[5902] = {X 480.7358, Y 53.5168, Z -1.3333, A 0.000, B 0.000, C 0.000 }
gfCNCPoint1[5903] = {X 481.3972, Y 54.5253, Z -1.3333, A 0.000, B 0.000, C 0.000 }
gfCNCPoint1[5904] = {X 481.8831, Y 55.6291, Z -1.3333, A 0.000, B 0.000, C 0.000 }
gfCNCPoint1[5905] = {X 482.1801, Y 56.7981, Z -1.3333, A 0.000, B 0.000, C 0.000 }
gfCNCPoint1[5906] = {X 482.2800, Y 58.0000, Z -1.3333, A 0.000, B 0.000, C 0.000 }
gfCNCPoint1[5907] = {X 482.2798, Y 58.9942, Z -1.3333, A 0.000, B 0.000, C 0.000 }
gfCNCPoint1[5908] = {X 482.1577, Y 60.2628, Z -1.3333, A 0.000, B 0.000, C 0.000 }
gfCNCPoint1[5909] = {X 481.8163, Y 61.4906, Z -1.3333, A 0.000, B 0.000, C 0.000 }
gfCNCPoint1[5910] = {X 481.2661, Y 62.6401, Z -1.3333, A 0.000, B 0.000, C 0.000 }
gfCNCPoint1[5911] = {X 480.5237, Y 63.6761, Z -1.3333, A 0.000, B 0.000, C 0.000 }
gfCNCPoint1[5912] = {X 479.6122, Y 64.5667, Z -1.3333, A 0.000, B 0.000, C 0.000 }
gfCNCPoint1[5913] = {X 478.5592, Y 65.2847, Z -1.3333, A 0.000, B 0.000, C 0.000 }
gfCNCPoint1[5914] = {X 478.5596, Y 90.7253, Z -1.3333, A 0.000, B 0.000, C 0.000 }
gfCNCPoint1[5915] = {X 479.5421, Y 91.3837, Z -1.3333, A 0.000, B 0.000, C 0.000 }
gfCNCPoint1[5916] = {X 480.4046, Y 92.1931, Z -1.3333, A 0.000, B 0.000, C 0.000 }
gfCNCPoint1[5917] = {X 481.1240, Y 93.1318, Z -1.3333, A 0.000, B 0.000, C 0.000 }
gfCNCPoint1[5918] = {X 481.6814, Y 94.1750, Z -1.3333, A 0.000, B 0.000, C 0.000 }
gfCNCPoint1[5919] = {X 482.0618, Y 95.2949, Z -1.3333, A 0.000, B 0.000, C 0.000 }
gfCNCPoint1[5920] = {X 507.6820, Y 95.2949, Z -1.3333, A 0.000, B 0.000, C 0.000 }
gfCNCPoint1[5921] = {X 507.6820, Y 97.6949, Z -1.3333, A 0.000, B 0.000, C 0.000 }
gfCNCPoint1[5922] = {X 597.6965, Y 97.6949, Z -1.3333, A 0.000, B 0.000, C 0.000 }
gfCNCPoint1[5923] = {X 597.6965, Y 51.8000, Z -1.3333, A 0.000, B 0.000, C 0.000 }
gfCNCPoint1[5924] = {X 593.5565, Y 51.8000, Z -1.3333, A 0.000, B 0.000, C 0.000 }
gfCNCPoint1[5925] = {X 592.3428, Y 51.6908, Z -1.3333, A 0.000, B 0.000, C 0.000 }
gfCNCPoint1[5926] = {X 591.1680, Y 51.3667, Z -1.3333, A 0.000, B 0.000, C 0.000 }
gfCNCPoint1[5927] = {X 590.0699, Y 50.8381, Z -1.3333, A 0.000, B 0.000, C 0.000 }
gfCNCPoint1[5928] = {X 589.0838, Y 50.1220, Z -1.3333, A 0.000, B 0.000, C 0.000 }
gfCNCPoint1[5929] = {X 588.4736, Y 49.5171, Z -1.3333, A 0.000, B 0.000, C 0.000 }
gfCNCPoint1[5930] = {X 587.9446, Y 48.8401, Z -1.3333, A 0.000, B 0.000, C 0.000 }
gfCNCPoint1[5931] = {X 587.5052, Y 48.1018, Z -1.3333, A 0.000, B 0.000, C 0.000 }
gfCNCPoint1[5932] = {X 587.0658, Y 48.8401, Z -1.3333, A 0.000, B 0.000, C 0.000 }
gfCNCPoint1[5933] = {X 586.5368, Y 49.5171, Z -1.3333, A 0.000, B 0.000, C 0.000 }
gfCNCPoint1[5934] = {X 585.9266, Y 50.1220, Z -1.3333, A 0.000, B 0.000, C 0.000 }
gfCNCPoint1[5935] = {X 585.1803, Y 50.6880, Z -1.3333, A 0.000, B 0.000, C 0.000 }
gfCNCPoint1[5936] = {X 584.3634, Y 51.1461, Z -1.3333, A 0.000, B 0.000, C 0.000 }
gfCNCPoint1[5937] = {X 583.3013, Y 51.5442, Z -1.3333, A 0.000, B 0.000, C 0.000 }
gfCNCPoint1[5938] = {X 582.1877, Y 51.7603, Z -1.3333, A 0.000, B 0.000, C 0.000 }
gfCNCPoint1[5939] = {X 581.0538, Y 51.7882, Z -1.3333, A 0.000, B 0.000, C 0.000 }
gfCNCPoint1[5940] = {X 579.9310, Y 51.6273, Z -1.3333, A 0.000, B 0.000, C 0.000 }
gfCNCPoint1[5941] = {X 578.8505, Y 51.2819, Z -1.3333, A 0.000, B 0.000, C 0.000 }
gfCNCPoint1[5942] = {X 577.8425, Y 50.7618, Z -1.3333, A 0.000, B 0.000, C 0.000 }
gfCNCPoint1[5943] = {X 576.9350, Y 50.0813, Z -1.3333, A 0.000, B 0.000, C 0.000 }
gfCNCPoint1[5944] = {X 576.3133, Y 49.4513, Z -1.3333, A 0.000, B 0.000, C 0.000 }
gfCNCPoint1[5945] = {X 575.7786, Y 48.7459, Z -1.3333, A 0.000, B 0.000, C 0.000 }
gfCNCPoint1[5946] = {X 575.3401, Y 47.9770, Z -1.3333, A 0.000, B 0.000, C 0.000 }
gfCNCPoint1[5947] = {X 574.9017, Y 48.7459, Z -1.3333, A 0.000, B 0.000, C 0.000 }
gfCNCPoint1[5948] = {X 574.3670, Y 49.4513, Z -1.3333, A 0.000, B 0.000, C 0.000 }
gfCNCPoint1[5949] = {X 573.7453, Y 50.0813, Z -1.3333, A 0.000, B 0.000, C 0.000 }
gfCNCPoint1[5950] = {X 572.7526, Y 50.8143, Z -1.3333, A 0.000, B 0.000, C 0.000 }
gfCNCPoint1[5951] = {X 571.6437, Y 51.3558, Z -1.3333, A 0.000, B 0.000, C 0.000 }
gfCNCPoint1[5952] = {X 570.4553, Y 51.6880, Z -1.3333, A 0.000, B 0.000, C 0.000 }
gfCNCPoint1[5953] = {X 569.2264, Y 51.8000, Z -1.3333, A 0.000, B 0.000, C 0.000 }
gfCNCPoint1[5954] = {X 562.4443, Y 51.8000, Z -1.3333, A 0.000, B 0.000, C 0.000 }
gfCNCPoint1[5955] = {X 561.2635, Y 51.6967, Z -1.3333, A 0.000, B 0.000, C 0.000 }
gfCNCPoint1[5956] = {X 560.1186, Y 51.3899, Z -1.3333, A 0.000, B 0.000, C 0.000 }
gfCNCPoint1[5957] = {X 559.0443, Y 50.8890, Z -1.3333, A 0.000, B 0.000, C 0.000 }
gfCNCPoint1[5958] = {X 558.0733, Y 50.2091, Z -1.3333, A 0.000, B 0.000, C 0.000 }
gfCNCPoint1[5959] = {X 557.2352, Y 49.3710, Z -1.3333, A 0.000, B 0.000, C 0.000 }
gfCNCPoint1[5960] = {X 556.5553, Y 48.4000, Z -1.3333, A 0.000, B 0.000, C 0.000 }
gfCNCPoint1[5961] = {X 556.0544, Y 47.3257, Z -1.3333, A 0.000, B 0.000, C 0.000 }
gfCNCPoint1[5962] = {X 555.7476, Y 46.1808, Z -1.3333, A 0.000, B 0.000, C 0.000 }
gfCNCPoint1[5963] = {X 555.6443, Y 45.0000, Z -1.3333, A 0.000, B 0.000, C 0.000 }
gfCNCPoint1[5964] = {X 555.6443, Y 44.0660, Z -1.3333, A 0.000, B 0.000, C 0.000 }
gfCNCPoint1[5965] = {X 555.7460, Y 42.9114, Z -1.3333, A 0.000, B 0.000, C 0.000 }
gfCNCPoint1[5966] = {X 556.0412, Y 41.7905, Z -1.3333, A 0.000, B 0.000, C 0.000 }
gfCNCPoint1[5967] = {X 556.5215, Y 40.7356, Z -1.3333, A 0.000, B 0.000, C 0.000 }
gfCNCPoint1[5968] = {X 557.1730, Y 39.7770, Z -1.3333, A 0.000, B 0.000, C 0.000 }
gfCNCPoint1[5969] = {X 557.1730, Y 10.2298, Z -1.3333, A 0.000, B 0.000, C 0.000 }
gfCNCPoint1[5970] = {X 556.5264, Y 9.2834, Z -1.3333, A 0.000, B 0.000, C 0.000 }
gfCNCPoint1[5971] = {X 556.0479, Y 8.2419, Z -1.3333, A 0.000, B 0.000, C 0.000 }
gfCNCPoint1[5972] = {X 555.7511, Y 7.1347, Z -1.3333, A 0.000, B 0.000, C 0.000 }
gfCNCPoint1[5973] = {X 555.6446, Y 5.9935, Z -1.3333, A 0.000, B 0.000, C 0.000 }
gfCNCPoint1[5974] = {X 555.6443, Y 5.0000, Z -1.3333, A 0.000, B 0.000, C 0.000 }
gfCNCPoint1[5975] = {X 555.6452, Y 4.8910, Z -1.3333, A 0.000, B 0.000, C 0.000 }
gfCNCPoint1[5976] = {X 555.6478, Y 4.7820, Z -1.3333, A 0.000, B 0.000, C 0.000 }
gfCNCPoint1[5977] = {X 555.8079, Y 3.5175, Z -1.3333, A 0.000, B 0.000, C 0.000 }
gfCNCPoint1[5978] = {X 556.2011, Y 2.3051, Z -1.3333, A 0.000, B 0.000, C 0.000 }
gfCNCPoint1[5979] = {X 358.2570, Y 2.3051, Z -1.3333, A 0.000, B 0.000, C 0.000 }
gfCNCPoint1[5980] = {X 360.1186, Y 3.4748, Z -1.3333, A 0.000, B 0.000, C 0.000 }
gfCNCPoint1[5981] = {X 361.8517, Y 4.8278, Z -1.3333, A 0.000, B 0.000, C 0.000 }
gfCNCPoint1[5982] = {X 363.4381, Y 6.3500, Z -1.3333, A 0.000, B 0.000, C 0.000 }
gfCNCPoint1[5983] = {X 363.7830, Y 6.7252, Z -1.3333, A 0.000, B 0.000, C 0.000 }
gfCNCPoint1[5984] = {X 364.1189, Y 7.1084, Z -1.3333, A 0.000, B 0.000, C 0.000 }
gfCNCPoint1[5985] = {X 365.6221, Y 9.0483, Z -1.3333, A 0.000, B 0.000, C 0.000 }
gfCNCPoint1[5986] = {X 366.9301, Y 11.1248, Z -1.3333, A 0.000, B 0.000, C 0.000 }
gfCNCPoint1[5987] = {X 368.0306, Y 13.3183, Z -1.3333, A 0.000, B 0.000, C 0.000 }
gfCNCPoint1[5988] = {X 368.9133, Y 15.6082, Z -1.3333, A 0.000, B 0.000, C 0.000 }
gfCNCPoint1[5989] = {X 369.5697, Y 17.9729, Z -1.3333, A 0.000, B 0.000, C 0.000 }
gfCNCPoint1[5990] = {X 370.0568, Y 20.6505, Z -1.3333, A 0.000, B 0.000, C 0.000 }
gfCNCPoint1[5991] = {X 370.3161, Y 23.3596, Z -1.3333, A 0.000, B 0.000, C 0.000 }
gfCNCPoint1[5992] = {X 370.3456, Y 26.0809, Z -1.3333, A 0.000, B 0.000, C 0.000 }
gfCNCPoint1[5993] = {X 370.1453, Y 28.7951, Z -1.3333, A 0.000, B 0.000, C 0.000 }
gfCNCPoint1[5994] = {X 369.7165, Y 31.4826, Z -1.3333, A 0.000, B 0.000, C 0.000 }
gfCNCPoint1[5995] = {X 369.1808, Y 33.6349, Z -1.3333, A 0.000, B 0.000, C 0.000 }
gfCNCPoint1[5996] = {X 368.4569, Y 35.7315, Z -1.3333, A 0.000, B 0.000, C 0.000 }
gfCNCPoint1[5997] = {X 367.5506, Y 37.7559, Z -1.3333, A 0.000, B 0.000, C 0.000 }
gfCNCPoint1[5998] = {X 366.4690, Y 39.6922, Z -1.3333, A 0.000, B 0.000, C 0.000 }
gfCNCPoint1[5999] = {X 365.2204, Y 41.5254, Z -1.3333, A 0.000, B 0.000, C 0.000 }
gfCNCPoint1[6000] = {X 363.9629, Y 43.0750, Z -1.3333, A 0.000, B 0.000, C 0.000 }
gfCNCPoint1[6001] = {X 362.5745, Y 44.5083, Z -1.3333, A 0.000, B 0.000, C 0.000 }
gfCNCPoint1[6002] = {X 361.0657, Y 45.8143, Z -1.3333, A 0.000, B 0.000, C 0.000 }
gfCNCPoint1[6003] = {X 359.4482, Y 46.9831, Z -1.3333, A 0.000, B 0.000, C 0.000 }
gfCNCPoint1[6004] = {X 357.7345, Y 48.0055, Z -1.3333, A 0.000, B 0.000, C 0.000 }
gfCNCPoint1[6005] = {X 355.7248, Y 48.9196, Z -1.3333, A 0.000, B 0.000, C 0.000 }
gfCNCPoint1[6006] = {X 353.6373, Y 49.6384, Z -1.3333, A 0.000, B 0.000, C 0.000 }
gfCNCPoint1[6007] = {X 351.4910, Y 50.1555, Z -1.3333, A 0.000, B 0.000, C 0.000 }
gfCNCPoint1[6008] = {X 349.3052, Y 50.4662, Z -1.3333, A 0.000, B 0.000, C 0.000 }
gfCNCPoint1[6009] = {X 347.0997, Y 50.5676, Z -1.3333, A 0.000, B 0.000, C 0.000 }
gfCNCPoint1[6010] = {X 344.9865, Y 50.5314, Z -1.3333, A 0.000, B 0.000, C 0.000 }
gfCNCPoint1[6011] = {X 342.8843, Y 50.3121, Z -1.3333, A 0.000, B 0.000, C 0.000 }
gfCNCPoint1[6012] = {X 340.8090, Y 49.9115, Z -1.3333, A 0.000, B 0.000, C 0.000 }
gfCNCPoint1[6013] = {X 338.7763, Y 49.3326, Z -1.3333, A 0.000, B 0.000, C 0.000 }
gfCNCPoint1[6014] = {X 336.8014, Y 48.5797, Z -1.3333, A 0.000, B 0.000, C 0.000 }
gfCNCPoint1[6015] = {X 334.8991, Y 47.6585, Z -1.3333, A 0.000, B 0.000, C 0.000 }
gfCNCPoint1[6016] = {X 333.3431, Y 46.7012, Z -1.3333, A 0.000, B 0.000, C 0.000 }
gfCNCPoint1[6017] = {X 331.8622, Y 45.6314, Z -1.3333, A 0.000, B 0.000, C 0.000 }
gfCNCPoint1[6018] = {X 330.4646, Y 44.4549, Z -1.3333, A 0.000, B 0.000, C 0.000 }
gfCNCPoint1[6019] = {X 329.4671, Y 44.4079, Z -1.3333, A 0.000, B 0.000, C 0.000 }
gfCNCPoint1[6020] = {X 328.5001, Y 44.1589, Z -1.3333, A 0.000, B 0.000, C 0.000 }
gfCNCPoint1[6021] = {X 327.6040, Y 43.7182, Z -1.3333, A 0.000, B 0.000, C 0.000 }
gfCNCPoint1[6022] = {X 326.8164, Y 43.1044, Z -1.3333, A 0.000, B 0.000, C 0.000 }
gfCNCPoint1[6023] = {X 326.1897, Y 42.4934, Z -1.3333, A 0.000, B 0.000, C 0.000 }
gfCNCPoint1[6024] = {X 325.5686, Y 41.7541, Z -1.3333, A 0.000, B 0.000, C 0.000 }
gfCNCPoint1[6025] = {X 325.1052, Y 40.9070, Z -1.3333, A 0.000, B 0.000, C 0.000 }
gfCNCPoint1[6026] = {X 324.8177, Y 39.9852, Z -1.3333, A 0.000, B 0.000, C 0.000 }
gfCNCPoint1[6027] = {X 324.7172, Y 39.0249, Z -1.3333, A 0.000, B 0.000, C 0.000 }
gfCNCPoint1[6028] = {X 324.8079, Y 38.0635, Z -1.3333, A 0.000, B 0.000, C 0.000 }
gfCNCPoint1[6029] = {X 325.0860, Y 37.1389, Z -1.3333, A 0.000, B 0.000, C 0.000 }
gfCNCPoint1[6030] = {X 325.5408, Y 36.2871, Z -1.3333, A 0.000, B 0.000, C 0.000 }
gfCNCPoint1[6031] = {X 329.7739, Y 29.9576, Z -1.3333, A 0.000, B 0.000, C 0.000 }
gfCNCPoint1[6032] = {X 330.4584, Y 29.1427, Z -1.3333, A 0.000, B 0.000, C 0.000 }
gfCNCPoint1[6033] = {X 331.3033, Y 28.4956, Z -1.3333, A 0.000, B 0.000, C 0.000 }
gfCNCPoint1[6034] = {X 332.2684, Y 28.0471, Z -1.3333, A 0.000, B 0.000, C 0.000 }
gfCNCPoint1[6035] = {X 333.3078, Y 27.8184, Z -1.3333, A 0.000, B 0.000, C 0.000 }
gfCNCPoint1[6036] = {X 334.3720, Y 27.8205, Z -1.3333, A 0.000, B 0.000, C 0.000 }
gfCNCPoint1[6037] = {X 335.4105, Y 28.0532, Z -1.3333, A 0.000, B 0.000, C 0.000 }
gfCNCPoint1[6038] = {X 336.3738, Y 28.5055, Z -1.3333, A 0.000, B 0.000, C 0.000 }
gfCNCPoint1[6039] = {X 337.2162, Y 29.1559, Z -1.3333, A 0.000, B 0.000, C 0.000 }
gfCNCPoint1[6040] = {X 337.8209, Y 29.7387, Z -1.3333, A 0.000, B 0.000, C 0.000 }
gfCNCPoint1[6041] = {X 338.4998, Y 30.5717, Z -1.3333, A 0.000, B 0.000, C 0.000 }
gfCNCPoint1[6042] = {X 338.9800, Y 31.5330, Z -1.3333, A 0.000, B 0.000, C 0.000 }
gfCNCPoint1[6043] = {X 339.2382, Y 32.5762, Z -1.3333, A 0.000, B 0.000, C 0.000 }
gfCNCPoint1[6044] = {X 339.2618, Y 33.6505, Z -1.3333, A 0.000, B 0.000, C 0.000 }
gfCNCPoint1[6045] = {X 339.9057, Y 34.2220, Z -1.3333, A 0.000, B 0.000, C 0.000 }
gfCNCPoint1[6046] = {X 340.5743, Y 34.7645, Z -1.3333, A 0.000, B 0.000, C 0.000 }
gfCNCPoint1[6047] = {X 341.8061, Y 35.5733, Z -1.3333, A 0.000, B 0.000, C 0.000 }
gfCNCPoint1[6048] = {X 343.1428, Y 36.1935, Z -1.3333, A 0.000, B 0.000, C 0.000 }
gfCNCPoint1[6049] = {X 344.5559, Y 36.6116, Z -1.3333, A 0.000, B 0.000, C 0.000 }
gfCNCPoint1[6050] = {X 346.0149, Y 36.8186, Z -1.3333, A 0.000, B 0.000, C 0.000 }
gfCNCPoint1[6051] = {X 347.4884, Y 36.8102, Z -1.3333, A 0.000, B 0.000, C 0.000 }
gfCNCPoint1[6052] = {X 348.8411, Y 36.6284, Z -1.3333, A 0.000, B 0.000, C 0.000 }
gfCNCPoint1[6053] = {X 350.1460, Y 36.2283, Z -1.3333, A 0.000, B 0.000, C 0.000 }
